KUKA KRL program: EPS_2_251806_MH45A_A_20260213065140.src

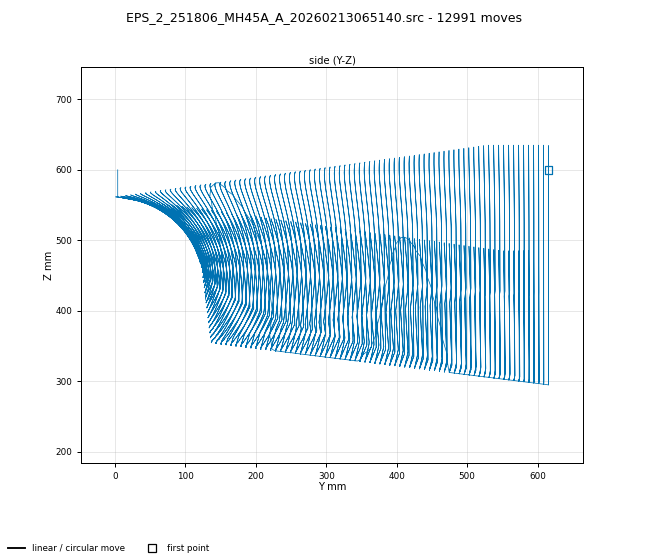
[picture p0: tool path of EPS_2_251806_MH45A_A_20260213065140.src, 12991 of 12993 moves have a stored position in this frame; points joined in program order, loops and branches not executed]
&ACCESS RVP
&REL 4
&COMMENT QRS 19112012
&PARAM EDITMASK = *
DEF PART()
EXT BAS (BAS_COMMAND :IN,REAL :IN )
INT I
BAS (#INITMOV,0 )

;KUKA QRS Post kuka4.cps  Date:22-06-2017 !

File_ID=3032

QRS_PRE_INIT()

;Init var - Until changes are made in qrs_pre_init
Outlet_Square_prg=0
Inlet_1_Square_prg=0
Inlet_2_Square_prg=0
Inlet_3_Square_prg=0
Inlet_4_Square_prg=0
Inlet_5_Square_prg=0

Outlet_1={X 0.000, Y 530.070, Z 534.500, B 0.000, E1 0.000 }
Inlet_1={X 0.000, Y 547.890, Z 284.500, B 0.000, E1 180.000 }
Outlet_1_type=201
Inlet_1_type=201
;QRS#1=Sidecore dimensions
;QRS#2=200-8" PVC SDR 35
;QRS#3=200-8" PVC SDR 35
;QRS#4=
;QRS#5=
;QRS#6=
;QRS#7=
;QRS#8=
;QRS#9=12-08 PSX
;QRS#10=12-08 PSX
;QRS#11=
;QRS#12=
;QRS#13=
;QRS#14=
;QRS#15=
;QRS#16=1220x127x914 3'
;QRS#17=EPS Height
;QRS#18=635
;QRS#19=*
;QRS#20= UPDATED VERSION 22-06-2017
;QRS#21=*
Outlet_Square=0100
Inlet_1_Square=0100
Inlet_2_Square=0
Inlet_3_Square=0
Inlet_4_Square=0
Inlet_5_Square=0
Mill_Square=1
Outlet_Square_Prg=204
Inlet_1_Square_prg=204

QRS_INIT()

$ADVANCE=5

; T1
PTP {E1 173.65,E2 173.65}
PTP {X 0,Y 615.429,A -85,B 0,C 180,E1 173.65,E2 173.65,E3 0,E4 0,E5 0,E6 0}
QRS_SPEED_INIT()
LIN {X 0,Y 615.429,Z 600,A -85,B 0,C 180,E1 173.65,E2 173.65,E3 0,E4 0,E5 0,E6 0} C_VEL
LIN {X 0,Y 615.429,Z 304.876,A -85,B 0,C 180,E1 173.65,E2 173.65} C_VEL
LIN {X 0,Y 615.429,Z 296.697,A -85,B 0,C 180,E1 173.65,E2 173.65} C_VEL
LIN {X 0,Y 615.425,Z 294.697,A -85,B 0,C 180,E1 173.464,E2 173.464} C_VEL
LIN {X 0,Y 615.464,Z 294.694,A -85,B 0,C 180,E1 170.801,E2 170.801} C_VEL
LIN {X 0,Y 615.465,Z 294.699,A -85,B 0,C 180,E1 168.139,E2 168.139} C_VEL
LIN {X 0,Y 615.424,Z 294.696,A -85,B 0,C 180,E1 165.449,E2 165.449} C_VEL
LIN {X 0,Y 615.48,Z 294.694,A -85,B 0,C 180,E1 162.729,E2 162.729} C_VEL
LIN {X 0,Y 615.442,Z 294.698,A -85,B 0,C 180,E1 159.966,E2 159.966} C_VEL
LIN {X 0,Y 615.425,Z 294.697,A -85,B 0,C 180,E1 157.666,E2 157.666} C_VEL
LIN {X 0,Y 615.425,Z 294.698,A -85,B 0,C 180,E1 155.725,E2 155.725} C_VEL
LIN {X 0,Y 615.424,Z 294.697,A -85,B 0,C 180,E1 153.553,E2 153.553} C_VEL
LIN {X 0,Y 615.493,Z 294.698,A -85,B 0,C 180,E1 150.594,E2 150.594} C_VEL
LIN {X 0,Y 615.472,Z 294.699,A -85,B 0,C 180,E1 148.314,E2 148.314} C_VEL
LIN {X 0,Y 615.436,Z 294.698,A -85,B 0,C 180,E1 145.975,E2 145.975} C_VEL
LIN {X 0,Y 615.423,Z 294.697,A -85,B 0,C 180,E1 143.571,E2 143.571} C_VEL
LIN {X 0,Y 615.464,Z 294.695,A -85,B 0,C 180,E1 140.939,E2 140.939} C_VEL
LIN {X 0,Y 615.495,Z 294.7,A -85,B 0,C 180,E1 138.527,E2 138.527} C_VEL
LIN {X 0,Y 615.426,Z 294.697,A -85,B 0,C 180,E1 135.845,E2 135.845} C_VEL
LIN {X 0,Y 615.459,Z 294.695,A -85,B 0,C 180,E1 133.044,E2 133.044} C_VEL
LIN {X 0,Y 615.437,Z 294.698,A -85,B 0,C 180,E1 130.083,E2 130.083} C_VEL
LIN {X 0,Y 615.429,Z 294.698,A -85,B 0,C 180,E1 128.005,E2 128.005} C_VEL
LIN {X 0,Y 615.42,Z 294.697,A -85,B 0,C 180,E1 125.62,E2 125.62} C_VEL
LIN {X 0,Y 615.445,Z 294.695,A -85,B 0,C 180,E1 123.238,E2 123.238} C_VEL
LIN {X 0,Y 615.486,Z 294.694,A -85,B 0,C 180,E1 120.919,E2 120.919} C_VEL
LIN {X 0,Y 615.465,Z 294.699,A -85,B 0,C 180,E1 118.446,E2 118.446} C_VEL
LIN {X 0,Y 615.463,Z 294.699,A -85,B 0,C 180,E1 116.445,E2 116.445} C_VEL
LIN {X 0,Y 615.424,Z 294.698,A -85,B 0,C 180,E1 113.994,E2 113.994} C_VEL
LIN {X 0,Y 615.433,Z 294.698,A -85,B 0,C 180,E1 112.138,E2 112.138} C_VEL
LIN {X 0,Y 615.425,Z 294.698,A -85,B 0,C 180,E1 110.034,E2 110.034} C_VEL
LIN {X 0,Y 615.423,Z 294.698,A -85,B 0,C 180,E1 107.959,E2 107.959} C_VEL
LIN {X 0,Y 615.422,Z 294.697,A -85,B 0,C 180,E1 105.907,E2 105.907} C_VEL
LIN {X 0,Y 615.458,Z 294.696,A -85,B 0,C 180,E1 103.202,E2 103.202} C_VEL
LIN {X 0,Y 615.498,Z 294.906,A -85,B 0,C 180,E1 102.676,E2 102.676} C_VEL
LIN {X 0,Y 615.497,Z 295.813,A -85,B 0,C 180,E1 102.572,E2 102.572} C_VEL
LIN {X 0,Y 615.497,Z 381.802,A -85,B 0,C 180,E1 101.526,E2 101.526} C_VEL
LIN {X 0,Y 615.498,Z 394.745,A -85,B 0,C 180,E1 101.234,E2 101.234} C_VEL
LIN {X 0,Y 615.498,Z 407.738,A -85,B 0,C 180,E1 100.8,E2 100.8} C_VEL
LIN {X 0,Y 615.496,Z 419.198,A -85,B 0,C 180,E1 100.277,E2 100.277} C_VEL
LIN {X 0,Y 615.492,Z 430.579,A -85,B 0,C 180,E1 99.613,E2 99.613} C_VEL
LIN {X 0,Y 615.498,Z 440.825,A -85,B 0,C 180,E1 98.867,E2 98.867} C_VEL
LIN {X 0,Y 615.499,Z 450.035,A -85,B 0,C 180,E1 98.04,E2 98.04} C_VEL
LIN {X 0,Y 615.499,Z 458.893,A -85,B 0,C 180,E1 97.057,E2 97.057} C_VEL
LIN {X 0,Y 615.497,Z 466.124,A -85,B 0,C 180,E1 96.063,E2 96.063} C_VEL
LIN {X 0,Y 615.497,Z 470.958,A -85,B 0,C 180,E1 95.241,E2 95.241} C_VEL
LIN {X 0,Y 615.494,Z 475.658,A -85,B 0,C 180,E1 94.256,E2 94.256} C_VEL
LIN {X 0,Y 615.494,Z 479.255,A -85,B 0,C 180,E1 93.273,E2 93.273} C_VEL
LIN {X 0,Y 615.496,Z 481.115,A -85,B 0,C 180,E1 92.618,E2 92.618} C_VEL
LIN {X 0,Y 615.499,Z 482.533,A -85,B 0,C 180,E1 91.963,E2 91.963} C_VEL
LIN {X 0,Y 615.496,Z 484.142,A -85,B 0,C 180,E1 90.654,E2 90.654} C_VEL
LIN {X 0,Y 615.495,Z 484.384,A -85,B 0,C 180,E1 90,E2 90} C_VEL
LIN {X 0,Y 615.495,Z 484.206,A -85,B 0,C 180,E1 89.346,E2 89.346} C_VEL
LIN {X 0,Y 615.499,Z 482.682,A -85,B 0,C 180,E1 88.037,E2 88.037} C_VEL
LIN {X 0,Y 615.498,Z 481.341,A -85,B 0,C 180,E1 87.382,E2 87.382} C_VEL
LIN {X 0,Y 615.496,Z 478.494,A -85,B 0,C 180,E1 86.399,E2 86.399} C_VEL
LIN {X 0,Y 615.498,Z 474.634,A -85,B 0,C 180,E1 85.416,E2 85.416} C_VEL
LIN {X 0,Y 615.498,Z 469.652,A -85,B 0,C 180,E1 84.43,E2 84.43} C_VEL
LIN {X 0,Y 615.496,Z 463.208,A -85,B 0,C 180,E1 83.418,E2 83.418} C_VEL
LIN {X 0,Y 615.497,Z 455.538,A -85,B 0,C 180,E1 82.455,E2 82.455} C_VEL
LIN {X 0,Y 615.498,Z 445.76,A -85,B 0,C 180,E1 81.464,E2 81.464} C_VEL
LIN {X 0,Y 615.498,Z 435.495,A -85,B 0,C 180,E1 80.636,E2 80.636} C_VEL
LIN {X 0,Y 615.495,Z 423.932,A -85,B 0,C 180,E1 79.889,E2 79.889} C_VEL
LIN {X 0,Y 615.499,Z 412.024,A -85,B 0,C 180,E1 79.291,E2 79.291} C_VEL
LIN {X 0,Y 615.498,Z 399.164,A -85,B 0,C 180,E1 78.807,E2 78.807} C_VEL
LIN {X 0,Y 615.497,Z 386.566,A -85,B 0,C 180,E1 78.474,E2 78.474} C_VEL
LIN {X 0,Y 615.498,Z 373.45,A -85,B 0,C 180,E1 78.265,E2 78.265} C_VEL
LIN {X 0,Y 615.498,Z 295.937,A -85,B 0,C 180,E1 77.345,E2 77.345} C_VEL
LIN {X 0,Y 615.498,Z 294.856,A -85,B 0,C 180,E1 77.219,E2 77.219} C_VEL
LIN {X 0,Y 615.454,Z 294.698,A -85,B 0,C 180,E1 74.773,E2 74.773} C_VEL
LIN {X 0,Y 615.447,Z 294.698,A -85,B 0,C 180,E1 72.729,E2 72.729} C_VEL
LIN {X 0,Y 615.436,Z 294.699,A -85,B 0,C 180,E1 70.661,E2 70.661} C_VEL
LIN {X 0,Y 615.43,Z 294.698,A -85,B 0,C 180,E1 68.566,E2 68.566} C_VEL
LIN {X 0,Y 615.422,Z 294.698,A -85,B 0,C 180,E1 66.441,E2 66.441} C_VEL
LIN {X 0,Y 615.414,Z 294.699,A -85,B 0,C 180,E1 64.281,E2 64.281} C_VEL
LIN {X 0,Y 615.415,Z 294.699,A -85,B 0,C 180,E1 62.082,E2 62.082} C_VEL
LIN {X 0,Y 615.428,Z 294.699,A -85,B 0,C 180,E1 59.837,E2 59.837} C_VEL
LIN {X 0,Y 615.459,Z 294.7,A -85,B 0,C 180,E1 57.541,E2 57.541} C_VEL
LIN {X 0,Y 615.498,Z 294.697,A -85,B 0,C 180,E1 55.186,E2 55.186} C_VEL
LIN {X 0,Y 615.44,Z 294.697,A -85,B 0,C 180,E1 52.755,E2 52.755} C_VEL
LIN {X 0,Y 615.416,Z 294.698,A -85,B 0,C 180,E1 50.245,E2 50.245} C_VEL
LIN {X 0,Y 615.454,Z 294.699,A -85,B 0,C 180,E1 47.645,E2 47.645} C_VEL
LIN {X 0,Y 615.454,Z 294.697,A -85,B 0,C 180,E1 44.929,E2 44.929} C_VEL
LIN {X 0,Y 615.467,Z 294.697,A -85,B 0,C 180,E1 43.046,E2 43.046} C_VEL
LIN {X 0,Y 615.425,Z 294.697,A -85,B 0,C 180,E1 40.612,E2 40.612} C_VEL
LIN {X 0,Y 615.428,Z 294.699,A -85,B 0,C 180,E1 38.006,E2 38.006} C_VEL
LIN {X 0,Y 615.468,Z 294.7,A -85,B 0,C 180,E1 35.617,E2 35.617} C_VEL
LIN {X 0,Y 615.483,Z 294.697,A -85,B 0,C 180,E1 33.237,E2 33.237} C_VEL
LIN {X 0,Y 615.445,Z 294.697,A -85,B 0,C 180,E1 30.922,E2 30.922} C_VEL
LIN {X 0,Y 615.419,Z 294.698,A -85,B 0,C 180,E1 28.44,E2 28.44} C_VEL
LIN {X 0,Y 615.419,Z 294.698,A -85,B 0,C 180,E1 26.447,E2 26.447} C_VEL
LIN {X 0,Y 615.435,Z 294.699,A -85,B 0,C 180,E1 24,E2 24} C_VEL
LIN {X 0,Y 615.498,Z 294.698,A -85,B 0,C 180,E1 21.432,E2 21.432} C_VEL
LIN {X 0,Y 615.421,Z 294.697,A -85,B 0,C 180,E1 18.589,E2 18.589} C_VEL
LIN {X 0,Y 615.42,Z 294.698,A -85,B 0,C 180,E1 16.413,E2 16.413} C_VEL
LIN {X 0,Y 615.451,Z 294.7,A -85,B 0,C 180,E1 13.875,E2 13.875} C_VEL
LIN {X 0,Y 615.464,Z 294.695,A -85,B 0,C 180,E1 11.194,E2 11.194} C_VEL
LIN {X 0,Y 615.421,Z 294.697,A -85,B 0,C 180,E1 8.538,E2 8.538} C_VEL
LIN {X 0,Y 615.454,Z 294.7,A -85,B 0,C 180,E1 5.899,E2 5.899} C_VEL
LIN {X 0,Y 615.469,Z 294.695,A -85,B 0,C 180,E1 3.273,E2 3.273} C_VEL
LIN {X 0,Y 615.422,Z 294.697,A -85,B 0,C 180,E1 0.654,E2 0.654} C_VEL
LIN {X 0,Y 615.45,Z 294.699,A -85,B 0,C 180,E1 -1.963,E2 -1.963} C_VEL
LIN {X 0,Y 615.483,Z 294.694,A -85,B 0,C 180,E1 -4.585,E2 -4.585} C_VEL
LIN {X 0,Y 615.423,Z 294.697,A -85,B 0,C 180,E1 -7.216,E2 -7.216} C_VEL
LIN {X 0,Y 615.425,Z 294.696,A -85,B 0,C 180,E1 -9.2,E2 -9.2} C_VEL
LIN {X 0,Y 615.424,Z 294.697,A -85,B 0,C 180,E1 -11.194,E2 -11.194} C_VEL
LIN {X 0,Y 615.424,Z 294.696,A -85,B 0,C 180,E1 -13.203,E2 -13.203} C_VEL
LIN {X 0,Y 615.422,Z 294.697,A -85,B 0,C 180,E1 -15.228,E2 -15.228} C_VEL
LIN {X 0,Y 615.422,Z 294.697,A -85,B 0,C 180,E1 -17.272,E2 -17.272} C_VEL
LIN {X 0,Y 615.423,Z 294.697,A -85,B 0,C 180,E1 -19.34,E2 -19.34} C_VEL
LIN {X 0,Y 615.425,Z 294.697,A -85,B 0,C 180,E1 -21.434,E2 -21.434} C_VEL
LIN {X 0,Y 615.473,Z 294.699,A -85,B 0,C 180,E1 -24.008,E2 -24.008} C_VEL
LIN {X 0,Y 615.486,Z 294.694,A -85,B 0,C 180,E1 -26.444,E2 -26.444} C_VEL
LIN {X 0,Y 615.456,Z 294.694,A -85,B 0,C 180,E1 -28.66,E2 -28.66} C_VEL
LIN {X 0,Y 615.427,Z 294.696,A -85,B 0,C 180,E1 -31.078,E2 -31.078} C_VEL
LIN {X 0,Y 615.425,Z 294.697,A -85,B 0,C 180,E1 -33.24,E2 -33.24} C_VEL
LIN {X 0,Y 615.458,Z 294.7,A -85,B 0,C 180,E1 -35.831,E2 -35.831} C_VEL
LIN {X 0,Y 615.487,Z 294.702,A -85,B 0,C 180,E1 -38.069,E2 -38.069} C_VEL
LIN {X 0,Y 615.455,Z 294.694,A -85,B 0,C 180,E1 -40.609,E2 -40.609} C_VEL
LIN {X 0,Y 615.427,Z 294.696,A -85,B 0,C 180,E1 -43.042,E2 -43.042} C_VEL
LIN {X 0,Y 615.426,Z 294.696,A -85,B 0,C 180,E1 -45.074,E2 -45.074} C_VEL
LIN {X 0,Y 615.45,Z 294.698,A -85,B 0,C 180,E1 -47.645,E2 -47.645} C_VEL
LIN {X 0,Y 615.491,Z 294.693,A -85,B 0,C 180,E1 -50.251,E2 -50.251} C_VEL
LIN {X 0,Y 615.437,Z 294.695,A -85,B 0,C 180,E1 -52.755,E2 -52.755} C_VEL
LIN {X 0,Y 615.427,Z 294.697,A -85,B 0,C 180,E1 -55.182,E2 -55.182} C_VEL
LIN {X 0,Y 615.46,Z 294.699,A -85,B 0,C 180,E1 -57.674,E2 -57.674} C_VEL
LIN {X 0,Y 615.447,Z 294.694,A -85,B 0,C 180,E1 -60.592,E2 -60.592} C_VEL
LIN {X 0,Y 615.426,Z 294.696,A -85,B 0,C 180,E1 -62.967,E2 -62.967} C_VEL
LIN {X 0,Y 615.497,Z 294.938,A -85,B 0,C 180,E1 -64.058,E2 -64.058} C_VEL
LIN {X 0,Y 615.487,Z 314.816,A -85,B 0,C 180,E1 -66.218,E2 -66.218} C_VEL
LIN {X 0,Y 615.493,Z 342.158,A -85,B 0,C 180,E1 -69.095,E2 -69.095} C_VEL
LIN {X 0,Y 615.484,Z 369.157,A -85,B 0,C 180,E1 -71.882,E2 -71.882} C_VEL
LIN {X 0,Y 615.477,Z 395.91,A -85,B 0,C 180,E1 -74.604,E2 -74.604} C_VEL
LIN {X 0,Y 615.498,Z 420.869,A -85,B 0,C 180,E1 -77.093,E2 -77.093} C_VEL
LIN {X 0,Y 615.486,Z 530.842,A -85,B 0,C 180,E1 -78.411,E2 -78.411} C_VEL
LIN {X 0,Y 615.499,Z 543.349,A -85,B 0,C 180,E1 -78.682,E2 -78.682} C_VEL
LIN {X 0,Y 615.496,Z 556.5,A -85,B 0,C 180,E1 -79.109,E2 -79.109} C_VEL
LIN {X 0,Y 615.482,Z 568.481,A -85,B 0,C 180,E1 -79.639,E2 -79.639} C_VEL
LIN {X 0,Y 615.487,Z 579.998,A -85,B 0,C 180,E1 -80.304,E2 -80.304} C_VEL
LIN {X 0,Y 615.499,Z 590.343,A -85,B 0,C 180,E1 -81.05,E2 -81.05} C_VEL
LIN {X 0,Y 615.497,Z 598.813,A -85,B 0,C 180,E1 -81.794,E2 -81.794} C_VEL
LIN {X 0,Y 615.498,Z 606.607,A -85,B 0,C 180,E1 -82.62,E2 -82.62} C_VEL
LIN {X 0,Y 615.496,Z 614.204,A -85,B 0,C 180,E1 -83.608,E2 -83.608} C_VEL
LIN {X 0,Y 615.498,Z 621.205,A -85,B 0,C 180,E1 -84.759,E2 -84.759} C_VEL
LIN {X 0,Y 615.493,Z 625.852,A -85,B 0,C 180,E1 -85.744,E2 -85.744} C_VEL
LIN {X 0,Y 615.495,Z 629.399,A -85,B 0,C 180,E1 -86.727,E2 -86.727} C_VEL
LIN {X 0,Y 615.497,Z 631.233,A -85,B 0,C 180,E1 -87.382,E2 -87.382} C_VEL
LIN {X 0,Y 615.497,Z 632.608,A -85,B 0,C 180,E1 -88.037,E2 -88.037} C_VEL
LIN {X 0,Y 615.496,Z 634.174,A -85,B 0,C 180,E1 -89.346,E2 -89.346} C_VEL
LIN {X 0,Y 615.494,Z 634.389,A -85,B 0,C 180,E1 -90,E2 -90} C_VEL
LIN {X 0,Y 615.496,Z 633.58,A -85,B 0,C 180,E1 -91.309,E2 -91.309} C_VEL
LIN {X 0,Y 615.497,Z 632.608,A -85,B 0,C 180,E1 -91.963,E2 -91.963} C_VEL
LIN {X 0,Y 615.497,Z 631.233,A -85,B 0,C 180,E1 -92.618,E2 -92.618} C_VEL
LIN {X 0,Y 615.496,Z 628.35,A -85,B 0,C 180,E1 -93.601,E2 -93.601} C_VEL
LIN {X 0,Y 615.498,Z 624.442,A -85,B 0,C 180,E1 -94.584,E2 -94.584} C_VEL
LIN {X 0,Y 615.499,Z 619.405,A -85,B 0,C 180,E1 -95.57,E2 -95.57} C_VEL
LIN {X 0,Y 615.497,Z 612.869,A -85,B 0,C 180,E1 -96.583,E2 -96.583} C_VEL
LIN {X 0,Y 615.497,Z 605.134,A -85,B 0,C 180,E1 -97.545,E2 -97.545} C_VEL
LIN {X 0,Y 615.498,Z 597.047,A -85,B 0,C 180,E1 -98.371,E2 -98.371} C_VEL
LIN {X 0,Y 615.499,Z 587.17,A -85,B 0,C 180,E1 -99.198,E2 -99.198} C_VEL
LIN {X 0,Y 615.488,Z 575.985,A -85,B 0,C 180,E1 -99.945,E2 -99.945} C_VEL
LIN {X 0,Y 615.486,Z 565.027,A -85,B 0,C 180,E1 -100.527,E2 -100.527} C_VEL
LIN {X 0,Y 615.499,Z 552.418,A -85,B 0,C 180,E1 -101.042,E2 -101.042} C_VEL
LIN {X 0,Y 615.498,Z 540.072,A -85,B 0,C 180,E1 -101.401,E2 -101.401} C_VEL
LIN {X 0,Y 615.484,Z 526.483,A -85,B 0,C 180,E1 -101.652,E2 -101.652} C_VEL
LIN {X 0,Y 615.498,Z 420.869,A -85,B 0,C 180,E1 -102.907,E2 -102.907} C_VEL
LIN {X 0,Y 615.477,Z 395.91,A -85,B 0,C 180,E1 -105.396,E2 -105.396} C_VEL
LIN {X 0,Y 615.484,Z 369.157,A -85,B 0,C 180,E1 -108.118,E2 -108.118} C_VEL
LIN {X 0,Y 615.493,Z 342.159,A -85,B 0,C 180,E1 -110.905,E2 -110.905} C_VEL
LIN {X 0,Y 615.487,Z 314.813,A -85,B 0,C 180,E1 -113.782,E2 -113.782} C_VEL
LIN {X 0,Y 615.495,Z 294.938,A -85,B 0,C 180,E1 -115.942,E2 -115.942} C_VEL
LIN {X 0,Y 615.43,Z 294.695,A -85,B 0,C 180,E1 -117.179,E2 -117.179} C_VEL
LIN {X 0,Y 615.494,Z 294.692,A -85,B 0,C 180,E1 -119.795,E2 -119.795} C_VEL
LIN {X 0,Y 615.448,Z 294.698,A -85,B 0,C 180,E1 -122.459,E2 -122.459} C_VEL
LIN {X 0,Y 615.428,Z 294.696,A -85,B 0,C 180,E1 -124.818,E2 -124.818} C_VEL
LIN {X 0,Y 615.437,Z 294.695,A -85,B 0,C 180,E1 -127.245,E2 -127.245} C_VEL
LIN {X 0,Y 615.485,Z 294.7,A -85,B 0,C 180,E1 -130.089,E2 -130.089} C_VEL
LIN {X 0,Y 615.451,Z 294.698,A -85,B 0,C 180,E1 -132.355,E2 -132.355} C_VEL
LIN {X 0,Y 615.427,Z 294.696,A -85,B 0,C 180,E1 -134.926,E2 -134.926} C_VEL
LIN {X 0,Y 615.428,Z 294.696,A -85,B 0,C 180,E1 -136.957,E2 -136.957} C_VEL
LIN {X 0,Y 615.456,Z 294.694,A -85,B 0,C 180,E1 -139.391,E2 -139.391} C_VEL
LIN {X 0,Y 615.479,Z 294.702,A -85,B 0,C 180,E1 -141.988,E2 -141.988} C_VEL
LIN {X 0,Y 615.443,Z 294.698,A -85,B 0,C 180,E1 -144.381,E2 -144.381} C_VEL
LIN {X 0,Y 615.426,Z 294.696,A -85,B 0,C 180,E1 -146.76,E2 -146.76} C_VEL
LIN {X 0,Y 615.435,Z 294.695,A -85,B 0,C 180,E1 -149.077,E2 -149.077} C_VEL
LIN {X 0,Y 615.484,Z 294.693,A -85,B 0,C 180,E1 -151.548,E2 -151.548} C_VEL
LIN {X 0,Y 615.446,Z 294.698,A -85,B 0,C 180,E1 -154.282,E2 -154.282} C_VEL
LIN {X 0,Y 615.434,Z 294.697,A -85,B 0,C 180,E1 -156.441,E2 -156.441} C_VEL
LIN {X 0,Y 615.428,Z 294.697,A -85,B 0,C 180,E1 -158.566,E2 -158.566} C_VEL
LIN {X 0,Y 615.426,Z 294.696,A -85,B 0,C 180,E1 -160.66,E2 -160.66} C_VEL
LIN {X 0,Y 615.471,Z 294.694,A -85,B 0,C 180,E1 -163.413,E2 -163.413} C_VEL
LIN {X 0,Y 615.453,Z 294.699,A -85,B 0,C 180,E1 -166.125,E2 -166.125} C_VEL
LIN {X 0,Y 615.451,Z 294.698,A -85,B 0,C 180,E1 -168.138,E2 -168.138} C_VEL
LIN {X 0,Y 615.45,Z 294.698,A -85,B 0,C 180,E1 -170.137,E2 -170.137} C_VEL
LIN {X 0,Y 615.45,Z 294.698,A -85,B 0,C 180,E1 -172.124,E2 -172.124} C_VEL
LIN {X 0,Y 615.451,Z 294.699,A -85,B 0,C 180,E1 -174.101,E2 -174.101} C_VEL
LIN {X 0,Y 615.453,Z 294.699,A -85,B 0,C 180,E1 -176.071,E2 -176.071} C_VEL
LIN {X 0,Y 615.455,Z 294.699,A -85,B 0,C 180,E1 -178.037,E2 -178.037} C_VEL
LIN {X 0,Y 615.425,Z 294.696,A -85,B 0,C 180,E1 -180.654,E2 -180.654} C_VEL
LIN {X 0,Y 615.469,Z 294.694,A -85,B 0,C 180,E1 -183.273,E2 -183.273} C_VEL
LIN {X 0,Y 615.465,Z 294.699,A -85,B 0,C 180,E1 -185.899,E2 -185.899} C_VEL
LIN {X 0,Y 615.425,Z 294.697,A -85,B 0,C 180,E1 -186.536,E2 -186.536} C_VEL
LIN {X 0,Y 614.774,Z 294.843,A -85,B 0,C 180,E1 -187.082,E2 -187.082} C_VEL
LIN {X 0,Y 611.963,Z 295.255,A -85,B 0,C 180,E1 -187.968,E2 -187.968} C_VEL
LIN {X 0,Y 609.573,Z 295.565,A -85,B 0,C 180,E1 -188.681,E2 -188.681} C_VEL
LIN {X 0,Y 608.533,Z 295.683,A -85,B 0,C 180,E1 -189.231,E2 -189.231} C_VEL
LIN {X 0,Y 608.441,Z 295.693,A -85,B 0,C 180,E1 -189.417,E2 -189.417} C_VEL
LIN {X 0,Y 608.434,Z 295.694,A -85,B 0,C 180,E1 -192,E2 -192} C_VEL
LIN {X 0,Y 608.4,Z 295.694,A -85,B 0,C 180,E1 -194.722,E2 -194.722} C_VEL
LIN {X 0,Y 608.438,Z 295.698,A -85,B 0,C 180,E1 -197.477,E2 -197.477} C_VEL
LIN {X 0,Y 608.413,Z 295.693,A -85,B 0,C 180,E1 -200.276,E2 -200.276} C_VEL
LIN {X 0,Y 608.42,Z 295.691,A -85,B 0,C 180,E1 -202.47,E2 -202.47} C_VEL
LIN {X 0,Y 608.436,Z 295.696,A -85,B 0,C 180,E1 -205.302,E2 -205.302} C_VEL
LIN {X 0,Y 608.426,Z 295.701,A -85,B 0,C 180,E1 -207.519,E2 -207.519} C_VEL
LIN {X 0,Y 608.417,Z 295.694,A -85,B 0,C 180,E1 -209.965,E2 -209.965} C_VEL
LIN {X 0,Y 608.407,Z 295.693,A -85,B 0,C 180,E1 -212.516,E2 -212.516} C_VEL
LIN {X 0,Y 608.41,Z 295.694,A -85,B 0,C 180,E1 -214.902,E2 -214.902} C_VEL
LIN {X 0,Y 608.438,Z 295.694,A -85,B 0,C 180,E1 -217.749,E2 -217.749} C_VEL
LIN {X 0,Y 608.396,Z 295.694,A -85,B 0,C 180,E1 -220.324,E2 -220.324} C_VEL
LIN {X 0,Y 608.394,Z 295.694,A -85,B 0,C 180,E1 -222.329,E2 -222.329} C_VEL
LIN {X 0,Y 608.404,Z 295.693,A -85,B 0,C 180,E1 -224.26,E2 -224.26} C_VEL
LIN {X 0,Y 608.427,Z 295.695,A -85,B 0,C 180,E1 -227.039,E2 -227.039} C_VEL
LIN {X 0,Y 608.435,Z 295.695,A -85,B 0,C 180,E1 -229.696,E2 -229.696} C_VEL
LIN {X 0,Y 608.401,Z 295.693,A -85,B 0,C 180,E1 -232.25,E2 -232.25} C_VEL
LIN {X 0,Y 608.454,Z 295.693,A -85,B 0,C 180,E1 -235.094,E2 -235.094} C_VEL
LIN {X 0,Y 608.428,Z 295.692,A -85,B 0,C 180,E1 -237.904,E2 -237.904} C_VEL
LIN {X 0,Y 608.41,Z 295.693,A -85,B 0,C 180,E1 -240.218,E2 -240.218} C_VEL
LIN {X 0,Y 608.436,Z 295.691,A -85,B 0,C 180,E1 -242.801,E2 -242.801} C_VEL
LIN {X 0,Y 608.429,Z 295.699,A -85,B 0,C 180,E1 -245.428,E2 -245.428} C_VEL
LIN {X 0,Y 608.421,Z 295.691,A -85,B 0,C 180,E1 -248.307,E2 -248.307} C_VEL
LIN {X 0,Y 608.406,Z 295.693,A -85,B 0,C 180,E1 -250.428,E2 -250.428} C_VEL
LIN {X 0,Y 608.413,Z 295.692,A -85,B 0,C 180,E1 -252.523,E2 -252.523} C_VEL
LIN {X 0,Y 608.426,Z 295.701,A -85,B 0,C 180,E1 -255.279,E2 -255.279} C_VEL
LIN {X 0,Y 608.496,Z 295.84,A -85,B 0,C 180,E1 -257.197,E2 -257.197} C_VEL
LIN {X 0,Y 608.589,Z 296.919,A -85,B 0,C 180,E1 -257.305,E2 -257.305} C_VEL
LIN {X 0,Y 608.558,Z 380.807,A -85,B 0,C 180,E1 -258.319,E2 -258.319} C_VEL
LIN {X 0,Y 608.538,Z 394.124,A -85,B 0,C 180,E1 -258.614,E2 -258.614} C_VEL
LIN {X 0,Y 608.529,Z 407.354,A -85,B 0,C 180,E1 -259.055,E2 -259.055} C_VEL
LIN {X 0,Y 608.508,Z 419.373,A -85,B 0,C 180,E1 -259.604,E2 -259.604} C_VEL
LIN {X 0,Y 608.506,Z 430.793,A -85,B 0,C 180,E1 -260.276,E2 -260.276} C_VEL
LIN {X 0,Y 608.474,Z 441.086,A -85,B 0,C 180,E1 -261.03,E2 -261.03} C_VEL
LIN {X 0,Y 608.464,Z 450.351,A -85,B 0,C 180,E1 -261.866,E2 -261.866} C_VEL
LIN {X 0,Y 608.466,Z 459.324,A -85,B 0,C 180,E1 -262.868,E2 -262.868} C_VEL
LIN {X 0,Y 608.444,Z 466.556,A -85,B 0,C 180,E1 -263.867,E2 -263.867} C_VEL
LIN {X 0,Y 608.462,Z 471.435,A -85,B 0,C 180,E1 -264.698,E2 -264.698} C_VEL
LIN {X 0,Y 608.439,Z 476.179,A -85,B 0,C 180,E1 -265.694,E2 -265.694} C_VEL
LIN {X 0,Y 608.425,Z 479.812,A -85,B 0,C 180,E1 -266.689,E2 -266.689} C_VEL
LIN {X 0,Y 608.425,Z 481.691,A -85,B 0,C 180,E1 -267.352,E2 -267.352} C_VEL
LIN {X 0,Y 608.444,Z 483.127,A -85,B 0,C 180,E1 -268.014,E2 -268.014} C_VEL
LIN {X 0,Y 608.439,Z 484.752,A -85,B 0,C 180,E1 -269.338,E2 -269.338} C_VEL
LIN {X 0,Y 608.435,Z 484.995,A -85,B 0,C 180,E1 -270,E2 -270} C_VEL
LIN {X 0,Y 608.438,Z 484.815,A -85,B 0,C 180,E1 -270.662,E2 -270.662} C_VEL
LIN {X 0,Y 608.444,Z 483.276,A -85,B 0,C 180,E1 -271.986,E2 -271.986} C_VEL
LIN {X 0,Y 608.426,Z 481.919,A -85,B 0,C 180,E1 -272.648,E2 -272.648} C_VEL
LIN {X 0,Y 608.449,Z 479.042,A -85,B 0,C 180,E1 -273.642,E2 -273.642} C_VEL
LIN {X 0,Y 608.433,Z 475.143,A -85,B 0,C 180,E1 -274.638,E2 -274.638} C_VEL
LIN {X 0,Y 608.45,Z 470.113,A -85,B 0,C 180,E1 -275.634,E2 -275.634} C_VEL
LIN {X 0,Y 608.441,Z 463.796,A -85,B 0,C 180,E1 -276.633,E2 -276.633} C_VEL
LIN {X 0,Y 608.475,Z 455.879,A -85,B 0,C 180,E1 -277.633,E2 -277.633} C_VEL
LIN {X 0,Y 608.472,Z 446.037,A -85,B 0,C 180,E1 -278.636,E2 -278.636} C_VEL
LIN {X 0,Y 608.48,Z 435.717,A -85,B 0,C 180,E1 -279.473,E2 -279.473} C_VEL
LIN {X 0,Y 608.492,Z 424.103,A -85,B 0,C 180,E1 -280.229,E2 -280.229} C_VEL
LIN {X 0,Y 608.529,Z 412.86,A -85,B 0,C 180,E1 -280.803,E2 -280.803} C_VEL
LIN {X 0,Y 608.538,Z 401.266,A -85,B 0,C 180,E1 -281.257,E2 -281.257} C_VEL
LIN {X 0,Y 608.539,Z 387.57,A -85,B 0,C 180,E1 -281.639,E2 -281.639} C_VEL
LIN {X 0,Y 608.573,Z 375.305,A -85,B 0,C 180,E1 -281.849,E2 -281.849} C_VEL
LIN {X 0,Y 608.593,Z 297.073,A -85,B 0,C 180,E1 -282.78,E2 -282.78} C_VEL
LIN {X 0,Y 608.507,Z 295.861,A -85,B 0,C 180,E1 -282.888,E2 -282.888} C_VEL
LIN {X 0,Y 608.431,Z 295.692,A -85,B 0,C 180,E1 -285.407,E2 -285.407} C_VEL
LIN {X 0,Y 608.395,Z 295.693,A -85,B 0,C 180,E1 -288.173,E2 -288.173} C_VEL
LIN {X 0,Y 608.44,Z 295.696,A -85,B 0,C 180,E1 -290.982,E2 -290.982} C_VEL
LIN {X 0,Y 608.425,Z 295.696,A -85,B 0,C 180,E1 -293.125,E2 -293.125} C_VEL
LIN {X 0,Y 608.394,Z 295.694,A -85,B 0,C 180,E1 -295.705,E2 -295.705} C_VEL
LIN {X 0,Y 608.404,Z 295.695,A -85,B 0,C 180,E1 -298.269,E2 -298.269} C_VEL
LIN {X 0,Y 608.433,Z 295.692,A -85,B 0,C 180,E1 -301.265,E2 -301.265} C_VEL
LIN {X 0,Y 608.395,Z 295.694,A -85,B 0,C 180,E1 -303.724,E2 -303.724} C_VEL
LIN {X 0,Y 608.424,Z 295.692,A -85,B 0,C 180,E1 -306.093,E2 -306.093} C_VEL
LIN {X 0,Y 608.413,Z 295.701,A -85,B 0,C 180,E1 -308.591,E2 -308.591} C_VEL
LIN {X 0,Y 608.416,Z 295.693,A -85,B 0,C 180,E1 -311.337,E2 -311.337} C_VEL
LIN {X 0,Y 608.417,Z 295.692,A -85,B 0,C 180,E1 -313.873,E2 -313.873} C_VEL
LIN {X 0,Y 608.48,Z 295.694,A -85,B 0,C 180,E1 -316.689,E2 -316.689} C_VEL
LIN {X 0,Y 608.442,Z 295.696,A -85,B 0,C 180,E1 -318.822,E2 -318.822} C_VEL
LIN {X 0,Y 608.396,Z 295.694,A -85,B 0,C 180,E1 -321.406,E2 -321.406} C_VEL
LIN {X 0,Y 608.423,Z 295.692,A -85,B 0,C 180,E1 -323.956,E2 -323.956} C_VEL
LIN {X 0,Y 608.436,Z 295.696,A -85,B 0,C 180,E1 -326.327,E2 -326.327} C_VEL
LIN {X 0,Y 608.435,Z 295.697,A -85,B 0,C 180,E1 -328.733,E2 -328.733} C_VEL
LIN {X 0,Y 608.418,Z 295.691,A -85,B 0,C 180,E1 -331.388,E2 -331.388} C_VEL
LIN {X 0,Y 608.402,Z 295.694,A -85,B 0,C 180,E1 -333.223,E2 -333.223} C_VEL
LIN {X 0,Y 608.405,Z 295.693,A -85,B 0,C 180,E1 -335.427,E2 -335.427} C_VEL
LIN {X 0,Y 608.453,Z 295.694,A -85,B 0,C 180,E1 -338.308,E2 -338.308} C_VEL
LIN {X 0,Y 608.407,Z 295.693,A -85,B 0,C 180,E1 -341.299,E2 -341.299} C_VEL
LIN {X 0,Y 608.415,Z 295.694,A -85,B 0,C 180,E1 -343.905,E2 -343.905} C_VEL
LIN {X 0,Y 608.441,Z 295.696,A -85,B 0,C 180,E1 -346.643,E2 -346.643} C_VEL
LIN {X 0,Y 608.406,Z 295.693,A -85,B 0,C 180,E1 -349.349,E2 -349.349} C_VEL
LIN {X 0,Y 608.402,Z 295.693,A -85,B 0,C 180,E1 -351.363,E2 -351.363} C_VEL
LIN {X 0,Y 608.425,Z 295.695,A -85,B 0,C 180,E1 -354.033,E2 -354.033} C_VEL
LIN {X 0,Y 608.462,Z 295.691,A -85,B 0,C 180,E1 -356.689,E2 -356.689} C_VEL
LIN {X 0,Y 608.401,Z 295.693,A -85,B 0,C 180,E1 -359.338,E2 -359.338} C_VEL
LIN {X 0,Y 608.412,Z 295.692,A -85,B 0,C 180,E1 -361.324,E2 -361.324} C_VEL
LIN {X 0,Y 608.394,Z 295.694,A -85,B 0,C 180,E1 -363.311,E2 -363.311} C_VEL
LIN {X 0,Y 608.425,Z 295.695,A -85,B 0,C 180,E1 -365.967,E2 -365.967} C_VEL
LIN {X 0,Y 608.442,Z 295.693,A -85,B 0,C 180,E1 -368.636,E2 -368.636} C_VEL
LIN {X 0,Y 608.403,Z 295.693,A -85,B 0,C 180,E1 -371.325,E2 -371.325} C_VEL
LIN {X 0,Y 608.443,Z 295.695,A -85,B 0,C 180,E1 -374.011,E2 -374.011} C_VEL
LIN {X 0,Y 608.421,Z 295.693,A -85,B 0,C 180,E1 -376.785,E2 -376.785} C_VEL
LIN {X 0,Y 608.41,Z 295.694,A -85,B 0,C 180,E1 -379.572,E2 -379.572} C_VEL
LIN {X 0,Y 608.469,Z 295.692,A -85,B 0,C 180,E1 -382.406,E2 -382.406} C_VEL
LIN {X 0,Y 608.435,Z 295.694,A -85,B 0,C 180,E1 -384.572,E2 -384.572} C_VEL
LIN {X 0,Y 608.414,Z 295.693,A -85,B 0,C 180,E1 -387.52,E2 -387.52} C_VEL
LIN {X 0,Y 608.47,Z 295.692,A -85,B 0,C 180,E1 -389.974,E2 -389.974} C_VEL
LIN {X 0,Y 608.425,Z 295.691,A -85,B 0,C 180,E1 -392.882,E2 -392.882} C_VEL
LIN {X 0,Y 608.402,Z 295.694,A -85,B 0,C 180,E1 -395.281,E2 -395.281} C_VEL
LIN {X 0,Y 608.46,Z 295.694,A -85,B 0,C 180,E1 -398.241,E2 -398.241} C_VEL
LIN {X 0,Y 608.397,Z 295.694,A -85,B 0,C 180,E1 -401.182,E2 -401.182} C_VEL
LIN {X 0,Y 608.422,Z 295.692,A -85,B 0,C 180,E1 -403.305,E2 -403.305} C_VEL
LIN {X 0,Y 608.462,Z 295.695,A -85,B 0,C 180,E1 -406.131,E2 -406.131} C_VEL
LIN {X 0,Y 608.406,Z 295.693,A -85,B 0,C 180,E1 -408.82,E2 -408.82} C_VEL
LIN {X 0,Y 608.453,Z 295.693,A -85,B 0,C 180,E1 -411.762,E2 -411.762} C_VEL
LIN {X 0,Y 608.416,Z 295.693,A -85,B 0,C 180,E1 -414.721,E2 -414.721} C_VEL
LIN {X 0,Y 608.428,Z 295.693,A -85,B 0,C 180,E1 -417.483,E2 -417.483} C_VEL
LIN {X 0,Y 608.478,Z 295.69,A -85,B 0,C 180,E1 -420.222,E2 -420.222} C_VEL
LIN {X 0,Y 608.399,Z 295.697,A -85,B 0,C 180,E1 -423.224,E2 -423.224} C_VEL
LIN {X 0,Y 608.498,Z 295.939,A -85,B 0,C 180,E1 -423.864,E2 -423.864} C_VEL
LIN {X 0,Y 608.724,Z 300.805,A -85,B 0,C 180,E1 -424.418,E2 -424.418} C_VEL
LIN {X 0,Y 608.656,Z 325.517,A -85,B 0,C 180,E1 -427.082,E2 -427.082} C_VEL
LIN {X 0,Y 608.597,Z 352.244,A -85,B 0,C 180,E1 -429.907,E2 -429.907} C_VEL
LIN {X 0,Y 608.549,Z 379.14,A -85,B 0,C 180,E1 -432.7,E2 -432.7} C_VEL
LIN {X 0,Y 608.515,Z 406.036,A -85,B 0,C 180,E1 -435.452,E2 -435.452} C_VEL
LIN {X 0,Y 608.531,Z 420.908,A -85,B 0,C 180,E1 -436.943,E2 -436.943} C_VEL
LIN {X 0,Y 608.538,Z 530.958,A -85,B 0,C 180,E1 -438.277,E2 -438.277} C_VEL
LIN {X 0,Y 608.545,Z 544.223,A -85,B 0,C 180,E1 -438.572,E2 -438.572} C_VEL
LIN {X 0,Y 608.544,Z 557.333,A -85,B 0,C 180,E1 -439.009,E2 -439.009} C_VEL
LIN {X 0,Y 608.503,Z 568.638,A -85,B 0,C 180,E1 -439.519,E2 -439.519} C_VEL
LIN {X 0,Y 608.48,Z 580.2,A -85,B 0,C 180,E1 -440.191,E2 -440.191} C_VEL
LIN {X 0,Y 608.485,Z 590.596,A -85,B 0,C 180,E1 -440.946,E2 -440.946} C_VEL
LIN {X 0,Y 608.475,Z 599.113,A -85,B 0,C 180,E1 -441.699,E2 -441.699} C_VEL
LIN {X 0,Y 608.471,Z 606.961,A -85,B 0,C 180,E1 -442.534,E2 -442.534} C_VEL
LIN {X 0,Y 608.461,Z 614.287,A -85,B 0,C 180,E1 -443.485,E2 -443.485} C_VEL
LIN {X 0,Y 608.45,Z 619.866,A -85,B 0,C 180,E1 -444.366,E2 -444.366} C_VEL
LIN {X 0,Y 608.432,Z 624.95,A -85,B 0,C 180,E1 -445.362,E2 -445.362} C_VEL
LIN {X 0,Y 608.449,Z 628.896,A -85,B 0,C 180,E1 -446.358,E2 -446.358} C_VEL
LIN {X 0,Y 608.425,Z 631.809,A -85,B 0,C 180,E1 -447.352,E2 -447.352} C_VEL
LIN {X 0,Y 608.442,Z 633.201,A -85,B 0,C 180,E1 -448.014,E2 -448.014} C_VEL
LIN {X 0,Y 608.438,Z 634.783,A -85,B 0,C 180,E1 -449.338,E2 -449.338} C_VEL
LIN {X 0,Y 608.434,Z 635,A -85,B 0,C 180,E1 -450,E2 -450} C_VEL
LIN {X 0,Y 608.448,Z 634.184,A -85,B 0,C 180,E1 -451.324,E2 -451.324} C_VEL
LIN {X 0,Y 608.443,Z 633.201,A -85,B 0,C 180,E1 -451.986,E2 -451.986} C_VEL
LIN {X 0,Y 608.425,Z 631.809,A -85,B 0,C 180,E1 -452.648,E2 -452.648} C_VEL
LIN {X 0,Y 608.449,Z 628.896,A -85,B 0,C 180,E1 -453.642,E2 -453.642} C_VEL
LIN {X 0,Y 608.432,Z 624.95,A -85,B 0,C 180,E1 -454.638,E2 -454.638} C_VEL
LIN {X 0,Y 608.437,Z 618.877,A -85,B 0,C 180,E1 -455.801,E2 -455.801} C_VEL
LIN {X 0,Y 608.462,Z 612.236,A -85,B 0,C 180,E1 -456.799,E2 -456.799} C_VEL
LIN {X 0,Y 608.455,Z 603.99,A -85,B 0,C 180,E1 -457.8,E2 -457.8} C_VEL
LIN {X 0,Y 608.472,Z 595.538,A -85,B 0,C 180,E1 -458.636,E2 -458.636} C_VEL
LIN {X 0,Y 608.471,Z 585.093,A -85,B 0,C 180,E1 -459.473,E2 -459.473} C_VEL
LIN {X 0,Y 608.495,Z 574.759,A -85,B 0,C 180,E1 -460.144,E2 -460.144} C_VEL
LIN {X 0,Y 608.522,Z 563.243,A -85,B 0,C 180,E1 -460.741,E2 -460.741} C_VEL
LIN {X 0,Y 608.533,Z 551.878,A -85,B 0,C 180,E1 -461.192,E2 -461.192} C_VEL
LIN {X 0,Y 608.554,Z 538.362,A -85,B 0,C 180,E1 -461.575,E2 -461.575} C_VEL
LIN {X 0,Y 608.547,Z 525.101,A -85,B 0,C 180,E1 -461.808,E2 -461.808} C_VEL
LIN {X 0,Y 608.531,Z 420.907,A -85,B 0,C 180,E1 -463.057,E2 -463.057} C_VEL
LIN {X 0,Y 608.532,Z 392.588,A -85,B 0,C 180,E1 -465.919,E2 -465.919} C_VEL
LIN {X 0,Y 608.59,Z 364.011,A -85,B 0,C 180,E1 -468.865,E2 -468.865} C_VEL
LIN {X 0,Y 608.624,Z 337.116,A -85,B 0,C 180,E1 -471.685,E2 -471.685} C_VEL
LIN {X 0,Y 608.703,Z 311.369,A -85,B 0,C 180,E1 -474.436,E2 -474.436} C_VEL
LIN {X 0,Y 608.681,Z 296.772,A -85,B 0,C 180,E1 -476.024,E2 -476.024} C_VEL
LIN {X 0,Y 608.47,Z 295.745,A -85,B 0,C 180,E1 -476.195,E2 -476.195} C_VEL
LIN {X 0,Y 608.4,Z 295.694,A -85,B 0,C 180,E1 -479.023,E2 -479.023} C_VEL
LIN {X 0,Y 608.43,Z 295.691,A -85,B 0,C 180,E1 -481.318,E2 -481.318} C_VEL
LIN {X 0,Y 608.444,Z 295.694,A -85,B 0,C 180,E1 -483.731,E2 -483.731} C_VEL
LIN {X 0,Y 608.44,Z 295.699,A -85,B 0,C 180,E1 -486.092,E2 -486.092} C_VEL
LIN {X 0,Y 608.403,Z 295.695,A -85,B 0,C 180,E1 -488.592,E2 -488.592} C_VEL
LIN {X 0,Y 608.426,Z 295.692,A -85,B 0,C 180,E1 -491.338,E2 -491.338} C_VEL
LIN {X 0,Y 608.439,Z 295.694,A -85,B 0,C 180,E1 -494.262,E2 -494.262} C_VEL
LIN {X 0,Y 608.423,Z 295.691,A -85,B 0,C 180,E1 -496.695,E2 -496.695} C_VEL
LIN {X 0,Y 608.398,Z 295.694,A -85,B 0,C 180,E1 -498.819,E2 -498.819} C_VEL
LIN {X 0,Y 608.459,Z 295.694,A -85,B 0,C 180,E1 -501.759,E2 -501.759} C_VEL
LIN {X 0,Y 608.404,Z 295.693,A -85,B 0,C 180,E1 -504.72,E2 -504.72} C_VEL
LIN {X 0,Y 608.453,Z 295.691,A -85,B 0,C 180,E1 -507.477,E2 -507.477} C_VEL
LIN {X 0,Y 608.441,Z 295.693,A -85,B 0,C 180,E1 -510.219,E2 -510.219} C_VEL
LIN {X 0,Y 608.409,Z 295.692,A -85,B 0,C 180,E1 -512.803,E2 -512.803} C_VEL
LIN {X 0,Y 608.436,Z 295.693,A -85,B 0,C 180,E1 -515.428,E2 -515.428} C_VEL
LIN {X 0,Y 608.435,Z 295.692,A -85,B 0,C 180,E1 -518.307,E2 -518.307} C_VEL
LIN {X 0,Y 608.413,Z 295.693,A -85,B 0,C 180,E1 -520.428,E2 -520.428} C_VEL
LIN {X 0,Y 608.422,Z 295.693,A -85,B 0,C 180,E1 -523.215,E2 -523.215} C_VEL
LIN {X 0,Y 608.444,Z 295.695,A -85,B 0,C 180,E1 -525.989,E2 -525.989} C_VEL
LIN {X 0,Y 608.406,Z 295.693,A -85,B 0,C 180,E1 -528.675,E2 -528.675} C_VEL
LIN {X 0,Y 608.442,Z 295.693,A -85,B 0,C 180,E1 -531.364,E2 -531.364} C_VEL
LIN {X 0,Y 608.429,Z 295.695,A -85,B 0,C 180,E1 -534.033,E2 -534.033} C_VEL
LIN {X 0,Y 608.397,Z 295.694,A -85,B 0,C 180,E1 -536.689,E2 -536.689} C_VEL
LIN {X 0,Y 608.465,Z 295.69,A -85,B 0,C 180,E1 -539.338,E2 -539.338} C_VEL
LIN {X 0,Y 608.425,Z 295.696,A -85,B 0,C 180,E1 -541.986,E2 -541.986} C_VEL
LIN {X 0,Y 608.429,Z 295.696,A -85,B 0,C 180,E1 -543.974,E2 -543.974} C_VEL
LIN {X 0,Y 608.423,Z 295.691,A -85,B 0,C 180,E1 -546.633,E2 -546.633} C_VEL
LIN {X 0,Y 608.45,Z 295.692,A -85,B 0,C 180,E1 -549.306,E2 -549.306} C_VEL
LIN {X 0,Y 608.441,Z 295.693,A -85,B 0,C 180,E1 -549.417,E2 -549.417} C_VEL
LIN {X 0,Y 607.757,Z 295.779,A -85,B 0,C 180,E1 -549.97,E2 -549.97} C_VEL
LIN {X 0,Y 604.907,Z 296.132,A -85,B 0,C 180,E1 -550.866,E2 -550.866} C_VEL
LIN {X 0,Y 602.503,Z 296.439,A -85,B 0,C 180,E1 -551.588,E2 -551.588} C_VEL
LIN {X 0,Y 601.46,Z 296.561,A -85,B 0,C 180,E1 -552.144,E2 -552.144} C_VEL
LIN {X 0,Y 601.368,Z 296.57,A -85,B 0,C 180,E1 -552.333,E2 -552.333} C_VEL
LIN {X 0,Y 601.377,Z 296.569,A -85,B 0,C 180,E1 -554.898,E2 -554.898} C_VEL
LIN {X 0,Y 601.374,Z 296.578,A -85,B 0,C 180,E1 -557.689,E2 -557.689} C_VEL
LIN {X 0,Y 601.379,Z 296.574,A -85,B 0,C 180,E1 -559.81,E2 -559.81} C_VEL
LIN {X 0,Y 601.391,Z 296.567,A -85,B 0,C 180,E1 -562.684,E2 -562.684} C_VEL
LIN {X 0,Y 601.425,Z 296.572,A -85,B 0,C 180,E1 -565.618,E2 -565.618} C_VEL
LIN {X 0,Y 601.355,Z 296.575,A -85,B 0,C 180,E1 -567.871,E2 -567.871} C_VEL
LIN {X 0,Y 601.39,Z 296.567,A -85,B 0,C 180,E1 -570.166,E2 -570.166} C_VEL
LIN {X 0,Y 601.382,Z 296.568,A -85,B 0,C 180,E1 -572.711,E2 -572.711} C_VEL
LIN {X 0,Y 601.369,Z 296.574,A -85,B 0,C 180,E1 -575.11,E2 -575.11} C_VEL
LIN {X 0,Y 601.424,Z 296.573,A -85,B 0,C 180,E1 -577.42,E2 -577.42} C_VEL
LIN {X 0,Y 601.37,Z 296.571,A -85,B 0,C 180,E1 -579.999,E2 -579.999} C_VEL
LIN {X 0,Y 601.355,Z 296.572,A -85,B 0,C 180,E1 -582.586,E2 -582.586} C_VEL
LIN {X 0,Y 601.362,Z 296.57,A -85,B 0,C 180,E1 -584.53,E2 -584.53} C_VEL
LIN {X 0,Y 601.377,Z 296.579,A -85,B 0,C 180,E1 -587.413,E2 -587.413} C_VEL
LIN {X 0,Y 601.38,Z 296.57,A -85,B 0,C 180,E1 -590.003,E2 -590.003} C_VEL
LIN {X 0,Y 601.384,Z 296.568,A -85,B 0,C 180,E1 -592.625,E2 -592.625} C_VEL
LIN {X 0,Y 601.41,Z 296.57,A -85,B 0,C 180,E1 -595.069,E2 -595.069} C_VEL
LIN {X 0,Y 601.417,Z 296.572,A -85,B 0,C 180,E1 -597.484,E2 -597.484} C_VEL
LIN {X 0,Y 601.369,Z 296.572,A -85,B 0,C 180,E1 -599.862,E2 -599.862} C_VEL
LIN {X 0,Y 601.356,Z 296.57,A -85,B 0,C 180,E1 -602.13,E2 -602.13} C_VEL
LIN {X 0,Y 601.372,Z 296.569,A -85,B 0,C 180,E1 -604.38,E2 -604.38} C_VEL
LIN {X 0,Y 601.401,Z 296.575,A -85,B 0,C 180,E1 -607.317,E2 -607.317} C_VEL
LIN {X 0,Y 601.414,Z 296.571,A -85,B 0,C 180,E1 -609.478,E2 -609.478} C_VEL
LIN {X 0,Y 601.379,Z 296.571,A -85,B 0,C 180,E1 -611.607,E2 -611.607} C_VEL
LIN {X 0,Y 601.405,Z 296.569,A -85,B 0,C 180,E1 -613.712,E2 -613.712} C_VEL
LIN {X 0,Y 601.425,Z 296.569,A -85,B 0,C 180,E1 -616.829,E2 -616.829} C_VEL
LIN {X 0,Y 601.473,Z 296.881,A -85,B 0,C 180,E1 -617.087,E2 -617.087} C_VEL
LIN {X 0,Y 601.664,Z 298.237,A -85,B 0,C 180,E1 -617.177,E2 -617.177} C_VEL
LIN {X 0,Y 601.63,Z 380.837,A -85,B 0,C 180,E1 -618.183,E2 -618.183} C_VEL
LIN {X 0,Y 601.602,Z 394.145,A -85,B 0,C 180,E1 -618.481,E2 -618.481} C_VEL
LIN {X 0,Y 601.566,Z 407.226,A -85,B 0,C 180,E1 -618.921,E2 -618.921} C_VEL
LIN {X 0,Y 601.514,Z 419.383,A -85,B 0,C 180,E1 -619.481,E2 -619.481} C_VEL
LIN {X 0,Y 601.474,Z 430.804,A -85,B 0,C 180,E1 -620.161,E2 -620.161} C_VEL
LIN {X 0,Y 601.438,Z 441.095,A -85,B 0,C 180,E1 -620.924,E2 -620.924} C_VEL
LIN {X 0,Y 601.411,Z 450.356,A -85,B 0,C 180,E1 -621.77,E2 -621.77} C_VEL
LIN {X 0,Y 601.388,Z 459.329,A -85,B 0,C 180,E1 -622.783,E2 -622.783} C_VEL
LIN {X 0,Y 601.376,Z 466.469,A -85,B 0,C 180,E1 -623.781,E2 -623.781} C_VEL
LIN {X 0,Y 601.373,Z 471.438,A -85,B 0,C 180,E1 -624.636,E2 -624.636} C_VEL
LIN {X 0,Y 601.354,Z 476.181,A -85,B 0,C 180,E1 -625.643,E2 -625.643} C_VEL
LIN {X 0,Y 601.344,Z 479.815,A -85,B 0,C 180,E1 -626.65,E2 -626.65} C_VEL
LIN {X 0,Y 601.324,Z 481.693,A -85,B 0,C 180,E1 -627.32,E2 -627.32} C_VEL
LIN {X 0,Y 601.343,Z 483.127,A -85,B 0,C 180,E1 -627.991,E2 -627.991} C_VEL
LIN {X 0,Y 601.339,Z 484.753,A -85,B 0,C 180,E1 -629.33,E2 -629.33} C_VEL
LIN {X 0,Y 601.336,Z 484.996,A -85,B 0,C 180,E1 -630,E2 -630} C_VEL
LIN {X 0,Y 601.339,Z 484.815,A -85,B 0,C 180,E1 -630.67,E2 -630.67} C_VEL
LIN {X 0,Y 601.343,Z 483.276,A -85,B 0,C 180,E1 -632.009,E2 -632.009} C_VEL
LIN {X 0,Y 601.326,Z 481.917,A -85,B 0,C 180,E1 -632.68,E2 -632.68} C_VEL
LIN {X 0,Y 601.368,Z 479.04,A -85,B 0,C 180,E1 -633.685,E2 -633.685} C_VEL
LIN {X 0,Y 601.337,Z 475.141,A -85,B 0,C 180,E1 -634.693,E2 -634.693} C_VEL
LIN {X 0,Y 601.373,Z 470.11,A -85,B 0,C 180,E1 -635.701,E2 -635.701} C_VEL
LIN {X 0,Y 601.382,Z 463.792,A -85,B 0,C 180,E1 -636.711,E2 -636.711} C_VEL
LIN {X 0,Y 601.396,Z 455.874,A -85,B 0,C 180,E1 -637.723,E2 -637.723} C_VEL
LIN {X 0,Y 601.436,Z 446.031,A -85,B 0,C 180,E1 -638.737,E2 -638.737} C_VEL
LIN {X 0,Y 601.45,Z 435.711,A -85,B 0,C 180,E1 -639.585,E2 -639.585} C_VEL
LIN {X 0,Y 601.498,Z 424.092,A -85,B 0,C 180,E1 -640.349,E2 -640.349} C_VEL
LIN {X 0,Y 601.551,Z 412.85,A -85,B 0,C 180,E1 -640.93,E2 -640.93} C_VEL
LIN {X 0,Y 601.564,Z 400.436,A -85,B 0,C 180,E1 -641.416,E2 -641.416} C_VEL
LIN {X 0,Y 601.602,Z 387.548,A -85,B 0,C 180,E1 -641.775,E2 -641.775} C_VEL
LIN {X 0,Y 601.642,Z 375.267,A -85,B 0,C 180,E1 -641.988,E2 -641.988} C_VEL
LIN {X 0,Y 601.637,Z 297.653,A -85,B 0,C 180,E1 -642.931,E2 -642.931} C_VEL
LIN {X 0,Y 601.417,Z 296.639,A -85,B 0,C 180,E1 -643.064,E2 -643.064} C_VEL
LIN {X 0,Y 601.37,Z 296.571,A -85,B 0,C 180,E1 -645.592,E2 -645.592} C_VEL
LIN {X 0,Y 601.37,Z 296.566,A -85,B 0,C 180,E1 -648.393,E2 -648.393} C_VEL
LIN {X 0,Y 601.382,Z 296.571,A -85,B 0,C 180,E1 -651.24,E2 -651.24} C_VEL
LIN {X 0,Y 601.36,Z 296.572,A -85,B 0,C 180,E1 -653.412,E2 -653.412} C_VEL
LIN {X 0,Y 601.349,Z 296.572,A -85,B 0,C 180,E1 -655.854,E2 -655.854} C_VEL
LIN {X 0,Y 601.414,Z 296.571,A -85,B 0,C 180,E1 -658.627,E2 -658.627} C_VEL
LIN {X 0,Y 601.374,Z 296.569,A -85,B 0,C 180,E1 -661.728,E2 -661.728} C_VEL
LIN {X 0,Y 601.396,Z 296.568,A -85,B 0,C 180,E1 -664.12,E2 -664.12} C_VEL
LIN {X 0,Y 601.387,Z 296.576,A -85,B 0,C 180,E1 -666.583,E2 -666.583} C_VEL
LIN {X 0,Y 601.379,Z 296.569,A -85,B 0,C 180,E1 -669.528,E2 -669.528} C_VEL
LIN {X 0,Y 601.371,Z 296.569,A -85,B 0,C 180,E1 -671.769,E2 -671.769} C_VEL
LIN {X 0,Y 601.394,Z 296.574,A -85,B 0,C 180,E1 -674.532,E2 -674.532} C_VEL
LIN {X 0,Y 601.356,Z 296.572,A -85,B 0,C 180,E1 -677.325,E2 -677.325} C_VEL
LIN {X 0,Y 601.378,Z 296.568,A -85,B 0,C 180,E1 -679.43,E2 -679.43} C_VEL
LIN {X 0,Y 601.345,Z 296.572,A -85,B 0,C 180,E1 -681.726,E2 -681.726} C_VEL
LIN {X 0,Y 601.374,Z 296.569,A -85,B 0,C 180,E1 -683.742,E2 -683.742} C_VEL
LIN {X 0,Y 601.402,Z 296.574,A -85,B 0,C 180,E1 -686.685,E2 -686.685} C_VEL
LIN {X 0,Y 601.382,Z 296.569,A -85,B 0,C 180,E1 -689.056,E2 -689.056} C_VEL
LIN {X 0,Y 601.379,Z 296.567,A -85,B 0,C 180,E1 -691.37,E2 -691.37} C_VEL
LIN {X 0,Y 601.365,Z 296.57,A -85,B 0,C 180,E1 -693.634,E2 -693.634} C_VEL
LIN {X 0,Y 601.387,Z 296.569,A -85,B 0,C 180,E1 -695.857,E2 -695.857} C_VEL
LIN {X 0,Y 601.387,Z 296.573,A -85,B 0,C 180,E1 -698.76,E2 -698.76} C_VEL
LIN {X 0,Y 601.352,Z 296.572,A -85,B 0,C 180,E1 -701.606,E2 -701.606} C_VEL
LIN {X 0,Y 601.38,Z 296.569,A -85,B 0,C 180,E1 -703.711,E2 -703.711} C_VEL
LIN {X 0,Y 601.39,Z 296.577,A -85,B 0,C 180,E1 -706.483,E2 -706.483} C_VEL
LIN {X 0,Y 601.368,Z 296.57,A -85,B 0,C 180,E1 -709.223,E2 -709.223} C_VEL
LIN {X 0,Y 601.39,Z 296.57,A -85,B 0,C 180,E1 -711.938,E2 -711.938} C_VEL
LIN {X 0,Y 601.407,Z 296.571,A -85,B 0,C 180,E1 -714.636,E2 -714.636} C_VEL
LIN {X 0,Y 601.39,Z 296.567,A -85,B 0,C 180,E1 -717.321,E2 -717.321} C_VEL
LIN {X 0,Y 601.415,Z 296.568,A -85,B 0,C 180,E1 -720,E2 -720} C_VEL
LIN {X 0,Y 601.429,Z 296.567,A -85,B 0,C 180,E1 -722.679,E2 -722.679} C_VEL
LIN {X 0,Y 601.376,Z 296.568,A -85,B 0,C 180,E1 -725.365,E2 -725.365} C_VEL
LIN {X 0,Y 601.356,Z 296.571,A -85,B 0,C 180,E1 -727.386,E2 -727.386} C_VEL
LIN {X 0,Y 601.406,Z 296.572,A -85,B 0,C 180,E1 -730.095,E2 -730.095} C_VEL
LIN {X 0,Y 601.393,Z 296.568,A -85,B 0,C 180,E1 -732.829,E2 -732.829} C_VEL
LIN {X 0,Y 601.371,Z 296.571,A -85,B 0,C 180,E1 -735.592,E2 -735.592} C_VEL
LIN {X 0,Y 601.359,Z 296.573,A -85,B 0,C 180,E1 -737.69,E2 -737.69} C_VEL
LIN {X 0,Y 601.417,Z 296.568,A -85,B 0,C 180,E1 -740.522,E2 -740.522} C_VEL
LIN {X 0,Y 601.364,Z 296.571,A -85,B 0,C 180,E1 -743.413,E2 -743.413} C_VEL
LIN {X 0,Y 601.38,Z 296.574,A -85,B 0,C 180,E1 -745.863,E2 -745.863} C_VEL
LIN {X 0,Y 601.409,Z 296.566,A -85,B 0,C 180,E1 -748.786,E2 -748.786} C_VEL
LIN {X 0,Y 601.4,Z 296.567,A -85,B 0,C 180,E1 -751.453,E2 -751.453} C_VEL
LIN {X 0,Y 601.407,Z 296.575,A -85,B 0,C 180,E1 -754.12,E2 -754.12} C_VEL
LIN {X 0,Y 601.37,Z 296.573,A -85,B 0,C 180,E1 -756.585,E2 -756.585} C_VEL
LIN {X 0,Y 601.372,Z 296.569,A -85,B 0,C 180,E1 -759.13,E2 -759.13} C_VEL
LIN {X 0,Y 601.412,Z 296.57,A -85,B 0,C 180,E1 -761.766,E2 -761.766} C_VEL
LIN {X 0,Y 601.393,Z 296.568,A -85,B 0,C 180,E1 -764.533,E2 -764.533} C_VEL
LIN {X 0,Y 601.355,Z 296.572,A -85,B 0,C 180,E1 -767.326,E2 -767.326} C_VEL
LIN {X 0,Y 601.395,Z 296.577,A -85,B 0,C 180,E1 -770.005,E2 -770.005} C_VEL
LIN {X 0,Y 601.391,Z 296.569,A -85,B 0,C 180,E1 -772.624,E2 -772.624} C_VEL
LIN {X 0,Y 601.365,Z 296.57,A -85,B 0,C 180,E1 -775.065,E2 -775.065} C_VEL
LIN {X 0,Y 601.399,Z 296.569,A -85,B 0,C 180,E1 -777.483,E2 -777.483} C_VEL
LIN {X 0,Y 601.406,Z 296.574,A -85,B 0,C 180,E1 -779.856,E2 -779.856} C_VEL
LIN {X 0,Y 601.373,Z 296.575,A -85,B 0,C 180,E1 -782.886,E2 -782.886} C_VEL
LIN {X 0,Y 601.406,Z 296.744,A -85,B 0,C 180,E1 -783.614,E2 -783.614} C_VEL
LIN {X 0,Y 601.984,Z 299.994,A -85,B 0,C 180,E1 -784.021,E2 -784.021} C_VEL
LIN {X 0,Y 601.83,Z 325.517,A -85,B 0,C 180,E1 -786.807,E2 -786.807} C_VEL
LIN {X 0,Y 601.739,Z 350.563,A -85,B 0,C 180,E1 -789.49,E2 -789.49} C_VEL
LIN {X 0,Y 601.624,Z 377.459,A -85,B 0,C 180,E1 -792.319,E2 -792.319} C_VEL
LIN {X 0,Y 601.543,Z 404.355,A -85,B 0,C 180,E1 -795.106,E2 -795.106} C_VEL
LIN {X 0,Y 601.517,Z 420.904,A -85,B 0,C 180,E1 -796.788,E2 -796.788} C_VEL
LIN {X 0,Y 601.668,Z 426.739,A -85,B 0,C 180,E1 -796.877,E2 -796.877} C_VEL
LIN {X 0,Y 601.605,Z 530.958,A -85,B 0,C 180,E1 -798.14,E2 -798.14} C_VEL
LIN {X 0,Y 601.587,Z 544.224,A -85,B 0,C 180,E1 -798.438,E2 -798.438} C_VEL
LIN {X 0,Y 601.549,Z 555.926,A -85,B 0,C 180,E1 -798.826,E2 -798.826} C_VEL
LIN {X 0,Y 601.517,Z 566.927,A -85,B 0,C 180,E1 -799.311,E2 -799.311} C_VEL
LIN {X 0,Y 601.479,Z 577.583,A -85,B 0,C 180,E1 -799.906,E2 -799.906} C_VEL
LIN {X 0,Y 601.446,Z 588.478,A -85,B 0,C 180,E1 -800.67,E2 -800.67} C_VEL
LIN {X 0,Y 601.429,Z 599.113,A -85,B 0,C 180,E1 -801.601,E2 -801.601} C_VEL
LIN {X 0,Y 601.418,Z 606.961,A -85,B 0,C 180,E1 -802.446,E2 -802.446} C_VEL
LIN {X 0,Y 601.37,Z 614.225,A -85,B 0,C 180,E1 -803.398,E2 -803.398} C_VEL
LIN {X 0,Y 601.372,Z 619.867,A -85,B 0,C 180,E1 -804.299,E2 -804.299} C_VEL
LIN {X 0,Y 601.337,Z 624.95,A -85,B 0,C 180,E1 -805.307,E2 -805.307} C_VEL
LIN {X 0,Y 601.367,Z 628.896,A -85,B 0,C 180,E1 -806.315,E2 -806.315} C_VEL
LIN {X 0,Y 601.325,Z 631.809,A -85,B 0,C 180,E1 -807.32,E2 -807.32} C_VEL
LIN {X 0,Y 601.341,Z 633.202,A -85,B 0,C 180,E1 -807.991,E2 -807.991} C_VEL
LIN {X 0,Y 601.339,Z 634.784,A -85,B 0,C 180,E1 -809.33,E2 -809.33} C_VEL
LIN {X 0,Y 601.335,Z 635,A -85,B 0,C 180,E1 -810,E2 -810} C_VEL
LIN {X 0,Y 601.348,Z 634.184,A -85,B 0,C 180,E1 -811.339,E2 -811.339} C_VEL
LIN {X 0,Y 601.341,Z 633.202,A -85,B 0,C 180,E1 -812.009,E2 -812.009} C_VEL
LIN {X 0,Y 601.325,Z 631.809,A -85,B 0,C 180,E1 -812.68,E2 -812.68} C_VEL
LIN {X 0,Y 601.367,Z 628.896,A -85,B 0,C 180,E1 -813.685,E2 -813.685} C_VEL
LIN {X 0,Y 601.337,Z 624.95,A -85,B 0,C 180,E1 -814.693,E2 -814.693} C_VEL
LIN {X 0,Y 601.372,Z 618.878,A -85,B 0,C 180,E1 -815.869,E2 -815.869} C_VEL
LIN {X 0,Y 601.382,Z 612.236,A -85,B 0,C 180,E1 -816.88,E2 -816.88} C_VEL
LIN {X 0,Y 601.4,Z 603.991,A -85,B 0,C 180,E1 -817.892,E2 -817.892} C_VEL
LIN {X 0,Y 601.436,Z 595.539,A -85,B 0,C 180,E1 -818.737,E2 -818.737} C_VEL
LIN {X 0,Y 601.442,Z 585.095,A -85,B 0,C 180,E1 -819.585,E2 -819.585} C_VEL
LIN {X 0,Y 601.473,Z 574.76,A -85,B 0,C 180,E1 -820.264,E2 -820.264} C_VEL
LIN {X 0,Y 601.537,Z 563.898,A -85,B 0,C 180,E1 -820.836,E2 -820.836} C_VEL
LIN {X 0,Y 601.565,Z 551.378,A -85,B 0,C 180,E1 -821.34,E2 -821.34} C_VEL
LIN {X 0,Y 601.598,Z 538.361,A -85,B 0,C 180,E1 -821.711,E2 -821.711} C_VEL
LIN {X 0,Y 601.614,Z 525.101,A -85,B 0,C 180,E1 -821.946,E2 -821.946} C_VEL
LIN {X 0,Y 601.575,Z 421.549,A -85,B 0,C 180,E1 -823.19,E2 -823.19} C_VEL
LIN {X 0,Y 601.517,Z 420.348,A -85,B 0,C 180,E1 -823.255,E2 -823.255} C_VEL
LIN {X 0,Y 601.589,Z 392.588,A -85,B 0,C 180,E1 -826.108,E2 -826.108} C_VEL
LIN {X 0,Y 601.69,Z 364.011,A -85,B 0,C 180,E1 -829.09,E2 -829.09} C_VEL
LIN {X 0,Y 601.775,Z 338.797,A -85,B 0,C 180,E1 -831.765,E2 -831.765} C_VEL
LIN {X 0,Y 601.891,Z 314.504,A -85,B 0,C 180,E1 -834.388,E2 -834.388} C_VEL
LIN {X 0,Y 601.957,Z 299.013,A -85,B 0,C 180,E1 -836.089,E2 -836.089} C_VEL
LIN {X 0,Y 601.416,Z 296.663,A -85,B 0,C 180,E1 -836.409,E2 -836.409} C_VEL
LIN {X 0,Y 601.392,Z 296.568,A -85,B 0,C 180,E1 -839.394,E2 -839.394} C_VEL
LIN {X 0,Y 601.388,Z 296.573,A -85,B 0,C 180,E1 -841.727,E2 -841.727} C_VEL
LIN {X 0,Y 601.406,Z 296.574,A -85,B 0,C 180,E1 -844.119,E2 -844.119} C_VEL
LIN {X 0,Y 601.37,Z 296.572,A -85,B 0,C 180,E1 -846.585,E2 -846.585} C_VEL
LIN {X 0,Y 601.378,Z 296.568,A -85,B 0,C 180,E1 -849.128,E2 -849.128} C_VEL
LIN {X 0,Y 601.411,Z 296.571,A -85,B 0,C 180,E1 -851.765,E2 -851.765} C_VEL
LIN {X 0,Y 601.393,Z 296.567,A -85,B 0,C 180,E1 -854.532,E2 -854.532} C_VEL
LIN {X 0,Y 601.381,Z 296.57,A -85,B 0,C 180,E1 -857.411,E2 -857.411} C_VEL
LIN {X 0,Y 601.389,Z 296.576,A -85,B 0,C 180,E1 -860.003,E2 -860.003} C_VEL
LIN {X 0,Y 601.384,Z 296.566,A -85,B 0,C 180,E1 -862.623,E2 -862.623} C_VEL
LIN {X 0,Y 601.37,Z 296.569,A -85,B 0,C 180,E1 -865.065,E2 -865.065} C_VEL
LIN {X 0,Y 601.422,Z 296.567,A -85,B 0,C 180,E1 -867.484,E2 -867.484} C_VEL
LIN {X 0,Y 601.443,Z 296.571,A -85,B 0,C 180,E1 -869.847,E2 -869.847} C_VEL
LIN {X 0,Y 601.365,Z 296.57,A -85,B 0,C 180,E1 -872.645,E2 -872.645} C_VEL
LIN {X 0,Y 601.429,Z 296.571,A -85,B 0,C 180,E1 -875.707,E2 -875.707} C_VEL
LIN {X 0,Y 601.393,Z 296.573,A -85,B 0,C 180,E1 -878.04,E2 -878.04} C_VEL
LIN {X 0,Y 601.379,Z 296.572,A -85,B 0,C 180,E1 -880.19,E2 -880.19} C_VEL
LIN {X 0,Y 601.391,Z 296.567,A -85,B 0,C 180,E1 -883.013,E2 -883.013} C_VEL
LIN {X 0,Y 601.391,Z 296.575,A -85,B 0,C 180,E1 -885.916,E2 -885.916} C_VEL
LIN {X 0,Y 601.387,Z 296.568,A -85,B 0,C 180,E1 -888.541,E2 -888.541} C_VEL
LIN {X 0,Y 601.397,Z 296.569,A -85,B 0,C 180,E1 -891.262,E2 -891.262} C_VEL
LIN {X 0,Y 601.385,Z 296.574,A -85,B 0,C 180,E1 -893.963,E2 -893.963} C_VEL
LIN {X 0,Y 601.378,Z 296.575,A -85,B 0,C 180,E1 -895.979,E2 -895.979} C_VEL
LIN {X 0,Y 601.398,Z 296.571,A -85,B 0,C 180,E1 -897.991,E2 -897.991} C_VEL
LIN {X 0,Y 601.42,Z 296.568,A -85,B 0,C 180,E1 -900,E2 -900} C_VEL
LIN {X 0,Y 601.391,Z 296.567,A -85,B 0,C 180,E1 -902.679,E2 -902.679} C_VEL
LIN {X 0,Y 601.41,Z 296.57,A -85,B 0,C 180,E1 -905.364,E2 -905.364} C_VEL
LIN {X 0,Y 601.416,Z 296.567,A -85,B 0,C 180,E1 -908.061,E2 -908.061} C_VEL
LIN {X 0,Y 601.391,Z 296.568,A -85,B 0,C 180,E1 -911,E2 -911} C_VEL
LIN {X 0,Y 601.368,Z 296.57,A -85,B 0,C 180,E1 -912.333,E2 -912.333} C_VEL
LIN {X 0,Y 600.686,Z 296.656,A -85,B 0,C 180,E1 -912.892,E2 -912.892} C_VEL
LIN {X 0,Y 597.836,Z 297.016,A -85,B 0,C 180,E1 -913.8,E2 -913.8} C_VEL
LIN {X 0,Y 595.438,Z 297.312,A -85,B 0,C 180,E1 -914.53,E2 -914.53} C_VEL
LIN {X 0,Y 594.409,Z 297.438,A -85,B 0,C 180,E1 -915.094,E2 -915.094} C_VEL
LIN {X 0,Y 594.325,Z 297.449,A -85,B 0,C 180,E1 -915.284,E2 -915.284} C_VEL
LIN {X 0,Y 594.32,Z 297.453,A -85,B 0,C 180,E1 -917.906,E2 -917.906} C_VEL
LIN {X 0,Y 594.367,Z 297.442,A -85,B 0,C 180,E1 -920.777,E2 -920.777} C_VEL
LIN {X 0,Y 594.339,Z 297.453,A -85,B 0,C 180,E1 -923.706,E2 -923.706} C_VEL
LIN {X 0,Y 594.345,Z 297.447,A -85,B 0,C 180,E1 -926.017,E2 -926.017} C_VEL
LIN {X 0,Y 594.361,Z 297.443,A -85,B 0,C 180,E1 -929,E2 -929} C_VEL
LIN {X 0,Y 594.361,Z 297.45,A -85,B 0,C 180,E1 -931.642,E2 -931.642} C_VEL
LIN {X 0,Y 594.35,Z 297.445,A -85,B 0,C 180,E1 -934.136,E2 -934.136} C_VEL
LIN {X 0,Y 594.368,Z 297.446,A -85,B 0,C 180,E1 -937.088,E2 -937.088} C_VEL
LIN {X 0,Y 594.332,Z 297.45,A -85,B 0,C 180,E1 -939.77,E2 -939.77} C_VEL
LIN {X 0,Y 594.323,Z 297.447,A -85,B 0,C 180,E1 -942.38,E2 -942.38} C_VEL
LIN {X 0,Y 594.31,Z 297.451,A -85,B 0,C 180,E1 -944.805,E2 -944.805} C_VEL
LIN {X 0,Y 594.338,Z 297.452,A -85,B 0,C 180,E1 -947.623,E2 -947.623} C_VEL
LIN {X 0,Y 594.347,Z 297.445,A -85,B 0,C 180,E1 -950.318,E2 -950.318} C_VEL
LIN {X 0,Y 594.348,Z 297.447,A -85,B 0,C 180,E1 -952.911,E2 -952.911} C_VEL
LIN {X 0,Y 594.353,Z 297.446,A -85,B 0,C 180,E1 -955.866,E2 -955.866} C_VEL
LIN {X 0,Y 594.338,Z 297.446,A -85,B 0,C 180,E1 -958.649,E2 -958.649} C_VEL
LIN {X 0,Y 594.374,Z 297.447,A -85,B 0,C 180,E1 -961.044,E2 -961.044} C_VEL
LIN {X 0,Y 594.338,Z 297.446,A -85,B 0,C 180,E1 -964.055,E2 -964.055} C_VEL
LIN {X 0,Y 594.343,Z 297.451,A -85,B 0,C 180,E1 -967.032,E2 -967.032} C_VEL
LIN {X 0,Y 594.347,Z 297.446,A -85,B 0,C 180,E1 -969.946,E2 -969.946} C_VEL
LIN {X 0,Y 594.318,Z 297.444,A -85,B 0,C 180,E1 -972.094,E2 -972.094} C_VEL
LIN {X 0,Y 594.33,Z 297.448,A -85,B 0,C 180,E1 -974.218,E2 -974.218} C_VEL
LIN {X 0,Y 594.435,Z 297.594,A -85,B 0,C 180,E1 -976.91,E2 -976.91} C_VEL
LIN {X 0,Y 594.64,Z 298.703,A -85,B 0,C 180,E1 -977.023,E2 -977.023} C_VEL
LIN {X 0,Y 594.686,Z 380.867,A -85,B 0,C 180,E1 -978.043,E2 -978.043} C_VEL
LIN {X 0,Y 594.636,Z 394.166,A -85,B 0,C 180,E1 -978.344,E2 -978.344} C_VEL
LIN {X 0,Y 594.595,Z 406.159,A -85,B 0,C 180,E1 -978.748,E2 -978.748} C_VEL
LIN {X 0,Y 594.553,Z 417.768,A -85,B 0,C 180,E1 -979.271,E2 -979.271} C_VEL
LIN {X 0,Y 594.486,Z 429.534,A -85,B 0,C 180,E1 -979.958,E2 -979.958} C_VEL
LIN {X 0,Y 594.414,Z 440.044,A -85,B 0,C 180,E1 -980.73,E2 -980.73} C_VEL
LIN {X 0,Y 594.384,Z 448.648,A -85,B 0,C 180,E1 -981.501,E2 -981.501} C_VEL
LIN {X 0,Y 594.347,Z 456.574,A -85,B 0,C 180,E1 -982.356,E2 -982.356} C_VEL
LIN {X 0,Y 594.305,Z 464.395,A -85,B 0,C 180,E1 -983.39,E2 -983.39} C_VEL
LIN {X 0,Y 594.289,Z 471.441,A -85,B 0,C 180,E1 -984.571,E2 -984.571} C_VEL
LIN {X 0,Y 594.27,Z 476.184,A -85,B 0,C 180,E1 -985.591,E2 -985.591} C_VEL
LIN {X 0,Y 594.267,Z 479.817,A -85,B 0,C 180,E1 -986.61,E2 -986.61} C_VEL
LIN {X 0,Y 594.225,Z 481.695,A -85,B 0,C 180,E1 -987.288,E2 -987.288} C_VEL
LIN {X 0,Y 594.242,Z 483.127,A -85,B 0,C 180,E1 -987.967,E2 -987.967} C_VEL
LIN {X 0,Y 594.24,Z 484.753,A -85,B 0,C 180,E1 -989.322,E2 -989.322} C_VEL
LIN {X 0,Y 594.236,Z 484.996,A -85,B 0,C 180,E1 -990,E2 -990} C_VEL
LIN {X 0,Y 594.239,Z 484.815,A -85,B 0,C 180,E1 -990.678,E2 -990.678} C_VEL
LIN {X 0,Y 594.242,Z 483.276,A -85,B 0,C 180,E1 -992.033,E2 -992.033} C_VEL
LIN {X 0,Y 594.226,Z 481.915,A -85,B 0,C 180,E1 -992.712,E2 -992.712} C_VEL
LIN {X 0,Y 594.289,Z 479.038,A -85,B 0,C 180,E1 -993.729,E2 -993.729} C_VEL
LIN {X 0,Y 594.242,Z 475.139,A -85,B 0,C 180,E1 -994.749,E2 -994.749} C_VEL
LIN {X 0,Y 594.299,Z 470.108,A -85,B 0,C 180,E1 -995.769,E2 -995.769} C_VEL
LIN {X 0,Y 594.316,Z 463.788,A -85,B 0,C 180,E1 -996.791,E2 -996.791} C_VEL
LIN {X 0,Y 594.346,Z 455.869,A -85,B 0,C 180,E1 -997.815,E2 -997.815} C_VEL
LIN {X 0,Y 594.381,Z 446.024,A -85,B 0,C 180,E1 -998.842,E2 -998.842} C_VEL
LIN {X 0,Y 594.433,Z 435.706,A -85,B 0,C 180,E1 -999.699,E2 -999.699} C_VEL
LIN {X 0,Y 594.516,Z 424.08,A -85,B 0,C 180,E1 -1000.472,E2 -1000.472} C_VEL
LIN {X 0,Y 594.541,Z 412.257,A -85,B 0,C 180,E1 -1001.086,E2 -1001.086} C_VEL
LIN {X 0,Y 594.612,Z 399.24,A -85,B 0,C 180,E1 -1001.591,E2 -1001.591} C_VEL
LIN {X 0,Y 594.668,Z 386.607,A -85,B 0,C 180,E1 -1001.936,E2 -1001.936} C_VEL
LIN {X 0,Y 594.702,Z 373.469,A -85,B 0,C 180,E1 -1002.152,E2 -1002.152} C_VEL
LIN {X 0,Y 594.679,Z 298.787,A -85,B 0,C 180,E1 -1003.063,E2 -1003.063} C_VEL
LIN {X 0,Y 594.395,Z 297.612,A -85,B 0,C 180,E1 -1003.178,E2 -1003.178} C_VEL
LIN {X 0,Y 594.324,Z 297.448,A -85,B 0,C 180,E1 -1005.782,E2 -1005.782} C_VEL
LIN {X 0,Y 594.369,Z 297.451,A -85,B 0,C 180,E1 -1008.924,E2 -1008.924} C_VEL
LIN {X 0,Y 594.338,Z 297.446,A -85,B 0,C 180,E1 -1011.504,E2 -1011.504} C_VEL
LIN {X 0,Y 594.329,Z 297.447,A -85,B 0,C 180,E1 -1013.706,E2 -1013.706} C_VEL
LIN {X 0,Y 594.346,Z 297.454,A -85,B 0,C 180,E1 -1016.701,E2 -1016.701} C_VEL
LIN {X 0,Y 594.368,Z 297.448,A -85,B 0,C 180,E1 -1018.999,E2 -1018.999} C_VEL
LIN {X 0,Y 594.349,Z 297.444,A -85,B 0,C 180,E1 -1021.638,E2 -1021.638} C_VEL
LIN {X 0,Y 594.369,Z 297.45,A -85,B 0,C 180,E1 -1024.58,E2 -1024.58} C_VEL
LIN {X 0,Y 594.345,Z 297.444,A -85,B 0,C 180,E1 -1027.602,E2 -1027.602} C_VEL
LIN {X 0,Y 594.349,Z 297.453,A -85,B 0,C 180,E1 -1030.568,E2 -1030.568} C_VEL
LIN {X 0,Y 594.335,Z 297.446,A -85,B 0,C 180,E1 -1033.301,E2 -1033.301} C_VEL
LIN {X 0,Y 594.329,Z 297.45,A -85,B 0,C 180,E1 -1036.163,E2 -1036.163} C_VEL
LIN {X 0,Y 594.353,Z 297.445,A -85,B 0,C 180,E1 -1039.18,E2 -1039.18} C_VEL
LIN {X 0,Y 594.34,Z 297.446,A -85,B 0,C 180,E1 -1042.056,E2 -1042.056} C_VEL
LIN {X 0,Y 594.312,Z 297.458,A -85,B 0,C 180,E1 -1044.68,E2 -1044.68} C_VEL
LIN {X 0,Y 594.361,Z 297.445,A -85,B 0,C 180,E1 -1047.09,E2 -1047.09} C_VEL
LIN {X 0,Y 594.339,Z 297.443,A -85,B 0,C 180,E1 -1049.678,E2 -1049.678} C_VEL
LIN {X 0,Y 594.306,Z 297.448,A -85,B 0,C 180,E1 -1051.769,E2 -1051.769} C_VEL
LIN {X 0,Y 594.348,Z 297.447,A -85,B 0,C 180,E1 -1054.054,E2 -1054.054} C_VEL
LIN {X 0,Y 594.317,Z 297.45,A -85,B 0,C 180,E1 -1057.031,E2 -1057.031} C_VEL
LIN {X 0,Y 594.364,Z 297.442,A -85,B 0,C 180,E1 -1059.223,E2 -1059.223} C_VEL
LIN {X 0,Y 594.317,Z 297.452,A -85,B 0,C 180,E1 -1062.094,E2 -1062.094} C_VEL
LIN {X 0,Y 594.33,Z 297.449,A -85,B 0,C 180,E1 -1064.921,E2 -1064.921} C_VEL
LIN {X 0,Y 594.333,Z 297.447,A -85,B 0,C 180,E1 -1067.71,E2 -1067.71} C_VEL
LIN {X 0,Y 594.34,Z 297.454,A -85,B 0,C 180,E1 -1070.471,E2 -1070.471} C_VEL
LIN {X 0,Y 594.325,Z 297.447,A -85,B 0,C 180,E1 -1073.362,E2 -1073.362} C_VEL
LIN {X 0,Y 594.325,Z 297.451,A -85,B 0,C 180,E1 -1075.931,E2 -1075.931} C_VEL
LIN {X 0,Y 594.363,Z 297.447,A -85,B 0,C 180,E1 -1078.645,E2 -1078.645} C_VEL
LIN {X 0,Y 594.408,Z 297.442,A -85,B 0,C 180,E1 -1080.677,E2 -1080.677} C_VEL
LIN {X 0,Y 594.303,Z 297.45,A -85,B 0,C 180,E1 -1083.39,E2 -1083.39} C_VEL
LIN {X 0,Y 594.344,Z 297.444,A -85,B 0,C 180,E1 -1085.428,E2 -1085.428} C_VEL
LIN {X 0,Y 594.33,Z 297.446,A -85,B 0,C 180,E1 -1087.474,E2 -1087.474} C_VEL
LIN {X 0,Y 594.366,Z 297.452,A -85,B 0,C 180,E1 -1090.216,E2 -1090.216} C_VEL
LIN {X 0,Y 594.336,Z 297.446,A -85,B 0,C 180,E1 -1092.984,E2 -1092.984} C_VEL
LIN {X 0,Y 594.345,Z 297.445,A -85,B 0,C 180,E1 -1095.079,E2 -1095.079} C_VEL
LIN {X 0,Y 594.329,Z 297.447,A -85,B 0,C 180,E1 -1097.195,E2 -1097.195} C_VEL
LIN {X 0,Y 594.353,Z 297.45,A -85,B 0,C 180,E1 -1100.055,E2 -1100.055} C_VEL
LIN {X 0,Y 594.339,Z 297.446,A -85,B 0,C 180,E1 -1102.968,E2 -1102.968} C_VEL
LIN {X 0,Y 594.315,Z 297.448,A -85,B 0,C 180,E1 -1105.196,E2 -1105.196} C_VEL
LIN {X 0,Y 594.334,Z 297.447,A -85,B 0,C 180,E1 -1107.519,E2 -1107.519} C_VEL
LIN {X 0,Y 594.378,Z 297.448,A -85,B 0,C 180,E1 -1110.328,E2 -1110.328} C_VEL
LIN {X 0,Y 594.367,Z 297.442,A -85,B 0,C 180,E1 -1112.951,E2 -1112.951} C_VEL
LIN {X 0,Y 594.308,Z 297.45,A -85,B 0,C 180,E1 -1115.412,E2 -1115.412} C_VEL
LIN {X 0,Y 594.364,Z 297.45,A -85,B 0,C 180,E1 -1117.943,E2 -1117.943} C_VEL
LIN {X 0,Y 594.35,Z 297.445,A -85,B 0,C 180,E1 -1120.82,E2 -1120.82} C_VEL
LIN {X 0,Y 594.337,Z 297.446,A -85,B 0,C 180,E1 -1123.302,E2 -1123.302} C_VEL
LIN {X 0,Y 594.34,Z 297.454,A -85,B 0,C 180,E1 -1126.164,E2 -1126.164} C_VEL
LIN {X 0,Y 594.361,Z 297.445,A -85,B 0,C 180,E1 -1128.535,E2 -1128.535} C_VEL
LIN {X 0,Y 594.358,Z 297.443,A -85,B 0,C 180,E1 -1131.299,E2 -1131.299} C_VEL
LIN {X 0,Y 594.34,Z 297.452,A -85,B 0,C 180,E1 -1133.755,E2 -1133.755} C_VEL
LIN {X 0,Y 594.35,Z 297.45,A -85,B 0,C 180,E1 -1136.238,E2 -1136.238} C_VEL
LIN {X 0,Y 594.354,Z 297.445,A -85,B 0,C 180,E1 -1138.649,E2 -1138.649} C_VEL
LIN {X 0,Y 594.335,Z 297.446,A -85,B 0,C 180,E1 -1141.051,E2 -1141.051} C_VEL
LIN {X 0,Y 594.37,Z 297.672,A -85,B 0,C 180,E1 -1143.387,E2 -1143.387} C_VEL
LIN {X 0,Y 595.233,Z 302.361,A -85,B 0,C 180,E1 -1143.97,E2 -1143.97} C_VEL
LIN {X 0,Y 595.027,Z 327.03,A -85,B 0,C 180,E1 -1146.692,E2 -1146.692} C_VEL
LIN {X 0,Y 594.832,Z 353.925,A -85,B 0,C 180,E1 -1149.602,E2 -1149.602} C_VEL
LIN {X 0,Y 594.678,Z 379.14,A -85,B 0,C 180,E1 -1152.283,E2 -1152.283} C_VEL
LIN {X 0,Y 594.565,Z 406.036,A -85,B 0,C 180,E1 -1155.103,E2 -1155.103} C_VEL
LIN {X 0,Y 594.553,Z 421.131,A -85,B 0,C 180,E1 -1156.641,E2 -1156.641} C_VEL
LIN {X 0,Y 594.755,Z 426.739,A -85,B 0,C 180,E1 -1156.722,E2 -1156.722} C_VEL
LIN {X 0,Y 594.684,Z 530.958,A -85,B 0,C 180,E1 -1158,E2 -1158} C_VEL
LIN {X 0,Y 594.64,Z 543.465,A -85,B 0,C 180,E1 -1158.28,E2 -1158.28} C_VEL
LIN {X 0,Y 594.595,Z 556.577,A -85,B 0,C 180,E1 -1158.719,E2 -1158.719} C_VEL
LIN {X 0,Y 594.539,Z 568.636,A -85,B 0,C 180,E1 -1159.27,E2 -1159.27} C_VEL
LIN {X 0,Y 594.469,Z 580.203,A -85,B 0,C 180,E1 -1159.958,E2 -1159.958} C_VEL
LIN {X 0,Y 594.413,Z 590.598,A -85,B 0,C 180,E1 -1160.73,E2 -1160.73} C_VEL
LIN {X 0,Y 594.383,Z 599.114,A -85,B 0,C 180,E1 -1161.501,E2 -1161.501} C_VEL
LIN {X 0,Y 594.347,Z 606.961,A -85,B 0,C 180,E1 -1162.356,E2 -1162.356} C_VEL
LIN {X 0,Y 594.282,Z 614.813,A -85,B 0,C 180,E1 -1163.408,E2 -1163.408} C_VEL
LIN {X 0,Y 594.289,Z 621.681,A -85,B 0,C 180,E1 -1164.571,E2 -1164.571} C_VEL
LIN {X 0,Y 594.27,Z 626.372,A -85,B 0,C 180,E1 -1165.591,E2 -1165.591} C_VEL
LIN {X 0,Y 594.267,Z 629.956,A -85,B 0,C 180,E1 -1166.61,E2 -1166.61} C_VEL
LIN {X 0,Y 594.226,Z 631.809,A -85,B 0,C 180,E1 -1167.288,E2 -1167.288} C_VEL
LIN {X 0,Y 594.24,Z 633.201,A -85,B 0,C 180,E1 -1167.967,E2 -1167.967} C_VEL
LIN {X 0,Y 594.239,Z 634.784,A -85,B 0,C 180,E1 -1169.322,E2 -1169.322} C_VEL
LIN {X 0,Y 594.236,Z 635,A -85,B 0,C 180,E1 -1170,E2 -1170} C_VEL
LIN {X 0,Y 594.247,Z 634.185,A -85,B 0,C 180,E1 -1171.355,E2 -1171.355} C_VEL
LIN {X 0,Y 594.24,Z 633.202,A -85,B 0,C 180,E1 -1172.033,E2 -1172.033} C_VEL
LIN {X 0,Y 594.226,Z 631.81,A -85,B 0,C 180,E1 -1172.712,E2 -1172.712} C_VEL
LIN {X 0,Y 594.288,Z 628.896,A -85,B 0,C 180,E1 -1173.729,E2 -1173.729} C_VEL
LIN {X 0,Y 594.242,Z 624.95,A -85,B 0,C 180,E1 -1174.749,E2 -1174.749} C_VEL
LIN {X 0,Y 594.304,Z 618.878,A -85,B 0,C 180,E1 -1175.939,E2 -1175.939} C_VEL
LIN {X 0,Y 594.308,Z 612.237,A -85,B 0,C 180,E1 -1176.962,E2 -1176.962} C_VEL
LIN {X 0,Y 594.359,Z 603.991,A -85,B 0,C 180,E1 -1177.986,E2 -1177.986} C_VEL
LIN {X 0,Y 594.382,Z 595.539,A -85,B 0,C 180,E1 -1178.842,E2 -1178.842} C_VEL
LIN {X 0,Y 594.427,Z 585.096,A -85,B 0,C 180,E1 -1179.699,E2 -1179.699} C_VEL
LIN {X 0,Y 594.486,Z 574.762,A -85,B 0,C 180,E1 -1180.386,E2 -1180.386} C_VEL
LIN {X 0,Y 594.561,Z 563.691,A -85,B 0,C 180,E1 -1180.975,E2 -1180.975} C_VEL
LIN {X 0,Y 594.6,Z 551.706,A -85,B 0,C 180,E1 -1181.464,E2 -1181.464} C_VEL
LIN {X 0,Y 594.643,Z 538.36,A -85,B 0,C 180,E1 -1181.85,E2 -1181.85} C_VEL
LIN {X 0,Y 594.691,Z 525.101,A -85,B 0,C 180,E1 -1182.087,E2 -1182.087} C_VEL
LIN {X 0,Y 594.604,Z 421.535,A -85,B 0,C 180,E1 -1183.347,E2 -1183.347} C_VEL
LIN {X 0,Y 594.48,Z 420.348,A -85,B 0,C 180,E1 -1183.415,E2 -1183.415} C_VEL
LIN {X 0,Y 594.635,Z 392.588,A -85,B 0,C 180,E1 -1186.302,E2 -1186.302} C_VEL
LIN {X 0,Y 594.765,Z 364.011,A -85,B 0,C 180,E1 -1189.321,E2 -1189.321} C_VEL
LIN {X 0,Y 594.937,Z 338.797,A -85,B 0,C 180,E1 -1192.028,E2 -1192.028} C_VEL
LIN {X 0,Y 595.157,Z 313.432,A -85,B 0,C 180,E1 -1194.801,E2 -1194.801} C_VEL
LIN {X 0,Y 595.222,Z 300.972,A -85,B 0,C 180,E1 -1196.187,E2 -1196.187} C_VEL
LIN {X 0,Y 594.366,Z 297.567,A -85,B 0,C 180,E1 -1196.641,E2 -1196.641} C_VEL
LIN {X 0,Y 594.335,Z 297.446,A -85,B 0,C 180,E1 -1199,E2 -1199} C_VEL
LIN {X 0,Y 594.366,Z 297.446,A -85,B 0,C 180,E1 -1201.64,E2 -1201.64} C_VEL
LIN {X 0,Y 594.349,Z 297.446,A -85,B 0,C 180,E1 -1204.581,E2 -1204.581} C_VEL
LIN {X 0,Y 594.358,Z 297.447,A -85,B 0,C 180,E1 -1207.604,E2 -1207.604} C_VEL
LIN {X 0,Y 594.347,Z 297.446,A -85,B 0,C 180,E1 -1210.568,E2 -1210.568} C_VEL
LIN {X 0,Y 594.334,Z 297.447,A -85,B 0,C 180,E1 -1213.301,E2 -1213.301} C_VEL
LIN {X 0,Y 594.338,Z 297.452,A -85,B 0,C 180,E1 -1216.162,E2 -1216.162} C_VEL
LIN {X 0,Y 594.357,Z 297.445,A -85,B 0,C 180,E1 -1218.534,E2 -1218.534} C_VEL
LIN {X 0,Y 594.358,Z 297.443,A -85,B 0,C 180,E1 -1221.298,E2 -1221.298} C_VEL
LIN {X 0,Y 594.338,Z 297.45,A -85,B 0,C 180,E1 -1223.754,E2 -1223.754} C_VEL
LIN {X 0,Y 594.353,Z 297.448,A -85,B 0,C 180,E1 -1226.237,E2 -1226.237} C_VEL
LIN {X 0,Y 594.35,Z 297.445,A -85,B 0,C 180,E1 -1228.648,E2 -1228.648} C_VEL
LIN {X 0,Y 594.367,Z 297.441,A -85,B 0,C 180,E1 -1231.043,E2 -1231.043} C_VEL
LIN {X 0,Y 594.347,Z 297.451,A -85,B 0,C 180,E1 -1234.054,E2 -1234.054} C_VEL
LIN {X 0,Y 594.358,Z 297.446,A -85,B 0,C 180,E1 -1236.295,E2 -1236.295} C_VEL
LIN {X 0,Y 594.388,Z 297.439,A -85,B 0,C 180,E1 -1239.224,E2 -1239.224} C_VEL
LIN {X 0,Y 594.323,Z 297.453,A -85,B 0,C 180,E1 -1242.094,E2 -1242.094} C_VEL
LIN {X 0,Y 594.337,Z 297.449,A -85,B 0,C 180,E1 -1244.218,E2 -1244.218} C_VEL
LIN {X 0,Y 594.345,Z 297.446,A -85,B 0,C 180,E1 -1246.32,E2 -1246.32} C_VEL
LIN {X 0,Y 594.343,Z 297.446,A -85,B 0,C 180,E1 -1249.094,E2 -1249.094} C_VEL
LIN {X 0,Y 594.348,Z 297.453,A -85,B 0,C 180,E1 -1251.842,E2 -1251.842} C_VEL
LIN {X 0,Y 594.342,Z 297.452,A -85,B 0,C 180,E1 -1253.891,E2 -1253.891} C_VEL
LIN {X 0,Y 594.333,Z 297.453,A -85,B 0,C 180,E1 -1255.931,E2 -1255.931} C_VEL
LIN {X 0,Y 594.371,Z 297.447,A -85,B 0,C 180,E1 -1257.967,E2 -1257.967} C_VEL
LIN {X 0,Y 594.389,Z 297.443,A -85,B 0,C 180,E1 -1260,E2 -1260} C_VEL
LIN {X 0,Y 594.362,Z 297.442,A -85,B 0,C 180,E1 -1262.711,E2 -1262.711} C_VEL
LIN {X 0,Y 594.373,Z 297.448,A -85,B 0,C 180,E1 -1265.428,E2 -1265.428} C_VEL
LIN {X 0,Y 594.36,Z 297.445,A -85,B 0,C 180,E1 -1268.158,E2 -1268.158} C_VEL
LIN {X 0,Y 594.357,Z 297.445,A -85,B 0,C 180,E1 -1271.062,E2 -1271.062} C_VEL
LIN {X 0,Y 594.355,Z 297.452,A -85,B 0,C 180,E1 -1273.68,E2 -1273.68} C_VEL
LIN {X 0,Y 594.325,Z 297.449,A -85,B 0,C 180,E1 -1275.284,E2 -1275.284} C_VEL
LIN {X 0,Y 593.653,Z 297.538,A -85,B 0,C 180,E1 -1275.85,E2 -1275.85} C_VEL
LIN {X 0,Y 590.787,Z 297.895,A -85,B 0,C 180,E1 -1276.768,E2 -1276.768} C_VEL
LIN {X 0,Y 588.374,Z 298.198,A -85,B 0,C 180,E1 -1277.506,E2 -1277.506} C_VEL
LIN {X 0,Y 587.349,Z 298.319,A -85,B 0,C 180,E1 -1278.076,E2 -1278.076} C_VEL
LIN {X 0,Y 587.272,Z 298.327,A -85,B 0,C 180,E1 -1278.269,E2 -1278.269} C_VEL
LIN {X 0,Y 587.323,Z 298.321,A -85,B 0,C 180,E1 -1281.038,E2 -1281.038} C_VEL
LIN {X 0,Y 587.278,Z 298.328,A -85,B 0,C 180,E1 -1284.009,E2 -1284.009} C_VEL
LIN {X 0,Y 587.292,Z 298.323,A -85,B 0,C 180,E1 -1286.281,E2 -1286.281} C_VEL
LIN {X 0,Y 587.332,Z 298.319,A -85,B 0,C 180,E1 -1289.132,E2 -1289.132} C_VEL
LIN {X 0,Y 587.307,Z 298.326,A -85,B 0,C 180,E1 -1291.831,E2 -1291.831} C_VEL
LIN {X 0,Y 587.319,Z 298.32,A -85,B 0,C 180,E1 -1294.345,E2 -1294.345} C_VEL
LIN {X 0,Y 587.325,Z 298.325,A -85,B 0,C 180,E1 -1297.609,E2 -1297.609} C_VEL
LIN {X 0,Y 587.286,Z 298.323,A -85,B 0,C 180,E1 -1300.257,E2 -1300.257} C_VEL
LIN {X 0,Y 587.29,Z 298.329,A -85,B 0,C 180,E1 -1303.117,E2 -1303.117} C_VEL
LIN {X 0,Y 587.291,Z 298.323,A -85,B 0,C 180,E1 -1306.047,E2 -1306.047} C_VEL
LIN {X 0,Y 587.3,Z 298.325,A -85,B 0,C 180,E1 -1308.929,E2 -1308.929} C_VEL
LIN {X 0,Y 587.304,Z 298.329,A -85,B 0,C 180,E1 -1311.519,E2 -1311.519} C_VEL
LIN {X 0,Y 587.274,Z 298.326,A -85,B 0,C 180,E1 -1314.099,E2 -1314.099} C_VEL
LIN {X 0,Y 587.307,Z 298.322,A -85,B 0,C 180,E1 -1316.602,E2 -1316.602} C_VEL
LIN {X 0,Y 587.302,Z 298.327,A -85,B 0,C 180,E1 -1319.032,E2 -1319.032} C_VEL
LIN {X 0,Y 587.296,Z 298.329,A -85,B 0,C 180,E1 -1321.402,E2 -1321.402} C_VEL
LIN {X 0,Y 587.293,Z 298.326,A -85,B 0,C 180,E1 -1323.833,E2 -1323.833} C_VEL
LIN {X 0,Y 587.294,Z 298.326,A -85,B 0,C 180,E1 -1326.741,E2 -1326.741} C_VEL
LIN {X 0,Y 587.309,Z 298.325,A -85,B 0,C 180,E1 -1329.695,E2 -1329.695} C_VEL
LIN {X 0,Y 587.278,Z 298.322,A -85,B 0,C 180,E1 -1331.872,E2 -1331.872} C_VEL
LIN {X 0,Y 587.289,Z 298.326,A -85,B 0,C 180,E1 -1334.024,E2 -1334.024} C_VEL
LIN {X 0,Y 587.372,Z 298.523,A -85,B 0,C 180,E1 -1336.772,E2 -1336.772} C_VEL
LIN {X 0,Y 587.655,Z 299.676,A -85,B 0,C 180,E1 -1336.88,E2 -1336.88} C_VEL
LIN {X 0,Y 587.832,Z 328.522,A -85,B 0,C 180,E1 -1337.244,E2 -1337.244} C_VEL
LIN {X 0,Y 587.742,Z 380.897,A -85,B 0,C 180,E1 -1337.899,E2 -1337.899} C_VEL
LIN {X 0,Y 587.704,Z 394.187,A -85,B 0,C 180,E1 -1338.205,E2 -1338.205} C_VEL
LIN {X 0,Y 587.629,Z 406.75,A -85,B 0,C 180,E1 -1338.635,E2 -1338.635} C_VEL
LIN {X 0,Y 587.57,Z 417.782,A -85,B 0,C 180,E1 -1339.142,E2 -1339.142} C_VEL
LIN {X 0,Y 587.477,Z 429.54,A -85,B 0,C 180,E1 -1339.837,E2 -1339.837} C_VEL
LIN {X 0,Y 587.393,Z 440.053,A -85,B 0,C 180,E1 -1340.618,E2 -1340.618} C_VEL
LIN {X 0,Y 587.323,Z 448.654,A -85,B 0,C 180,E1 -1341.398,E2 -1341.398} C_VEL
LIN {X 0,Y 587.274,Z 456.579,A -85,B 0,C 180,E1 -1342.263,E2 -1342.263} C_VEL
LIN {X 0,Y 587.235,Z 463.149,A -85,B 0,C 180,E1 -1343.127,E2 -1343.127} C_VEL
LIN {X 0,Y 587.237,Z 469.619,A -85,B 0,C 180,E1 -1344.161,E2 -1344.161} C_VEL
LIN {X 0,Y 587.147,Z 474.759,A -85,B 0,C 180,E1 -1345.194,E2 -1345.194} C_VEL
LIN {X 0,Y 587.213,Z 478.748,A -85,B 0,C 180,E1 -1346.226,E2 -1346.226} C_VEL
LIN {X 0,Y 587.131,Z 481.698,A -85,B 0,C 180,E1 -1347.256,E2 -1347.256} C_VEL
LIN {X 0,Y 587.14,Z 483.127,A -85,B 0,C 180,E1 -1347.942,E2 -1347.942} C_VEL
LIN {X 0,Y 587.14,Z 484.754,A -85,B 0,C 180,E1 -1349.314,E2 -1349.314} C_VEL
LIN {X 0,Y 587.137,Z 484.996,A -85,B 0,C 180,E1 -1350,E2 -1350} C_VEL
LIN {X 0,Y 587.14,Z 484.815,A -85,B 0,C 180,E1 -1350.686,E2 -1350.686} C_VEL
LIN {X 0,Y 587.141,Z 483.274,A -85,B 0,C 180,E1 -1352.058,E2 -1352.058} C_VEL
LIN {X 0,Y 587.133,Z 481.914,A -85,B 0,C 180,E1 -1352.744,E2 -1352.744} C_VEL
LIN {X 0,Y 587.213,Z 479.036,A -85,B 0,C 180,E1 -1353.774,E2 -1353.774} C_VEL
LIN {X 0,Y 587.147,Z 475.136,A -85,B 0,C 180,E1 -1354.806,E2 -1354.806} C_VEL
LIN {X 0,Y 587.229,Z 470.105,A -85,B 0,C 180,E1 -1355.839,E2 -1355.839} C_VEL
LIN {X 0,Y 587.23,Z 463.785,A -85,B 0,C 180,E1 -1356.874,E2 -1356.874} C_VEL
LIN {X 0,Y 587.288,Z 455.865,A -85,B 0,C 180,E1 -1357.91,E2 -1357.91} C_VEL
LIN {X 0,Y 587.343,Z 446.018,A -85,B 0,C 180,E1 -1358.949,E2 -1358.949} C_VEL
LIN {X 0,Y 587.421,Z 435.701,A -85,B 0,C 180,E1 -1359.816,E2 -1359.816} C_VEL
LIN {X 0,Y 587.531,Z 424.068,A -85,B 0,C 180,E1 -1360.598,E2 -1360.598} C_VEL
LIN {X 0,Y 587.575,Z 413.282,A -85,B 0,C 180,E1 -1361.172,E2 -1361.172} C_VEL
LIN {X 0,Y 587.632,Z 400.594,A -85,B 0,C 180,E1 -1361.685,E2 -1361.685} C_VEL
LIN {X 0,Y 587.716,Z 387.501,A -85,B 0,C 180,E1 -1362.057,E2 -1362.057} C_VEL
LIN {X 0,Y 587.785,Z 375.188,A -85,B 0,C 180,E1 -1362.275,E2 -1362.275} C_VEL
LIN {X 0,Y 587.762,Z 300.193,A -85,B 0,C 180,E1 -1363.197,E2 -1363.197} C_VEL
LIN {X 0,Y 587.408,Z 298.821,A -85,B 0,C 180,E1 -1363.271,E2 -1363.271} C_VEL
LIN {X 0,Y 587.302,Z 298.35,A -85,B 0,C 180,E1 -1363.406,E2 -1363.406} C_VEL
LIN {X 0,Y 587.283,Z 298.326,A -85,B 0,C 180,E1 -1365.976,E2 -1365.976} C_VEL
LIN {X 0,Y 587.315,Z 298.328,A -85,B 0,C 180,E1 -1369.031,E2 -1369.031} C_VEL
LIN {X 0,Y 587.295,Z 298.322,A -85,B 0,C 180,E1 -1371.775,E2 -1371.775} C_VEL
LIN {X 0,Y 587.282,Z 298.331,A -85,B 0,C 180,E1 -1374.564,E2 -1374.564} C_VEL
LIN {X 0,Y 587.293,Z 298.326,A -85,B 0,C 180,E1 -1377.048,E2 -1377.048} C_VEL
LIN {X 0,Y 587.299,Z 298.324,A -85,B 0,C 180,E1 -1379.382,E2 -1379.382} C_VEL
LIN {X 0,Y 587.313,Z 298.321,A -85,B 0,C 180,E1 -1381.83,E2 -1381.83} C_VEL
LIN {X 0,Y 587.326,Z 298.323,A -85,B 0,C 180,E1 -1384.344,E2 -1384.344} C_VEL
LIN {X 0,Y 587.3,Z 298.321,A -85,B 0,C 180,E1 -1387.61,E2 -1387.61} C_VEL
LIN {X 0,Y 587.291,Z 298.327,A -85,B 0,C 180,E1 -1390.255,E2 -1390.255} C_VEL
LIN {X 0,Y 587.282,Z 298.326,A -85,B 0,C 180,E1 -1393.114,E2 -1393.114} C_VEL
LIN {X 0,Y 587.281,Z 298.326,A -85,B 0,C 180,E1 -1396.045,E2 -1396.045} C_VEL
LIN {X 0,Y 587.303,Z 298.326,A -85,B 0,C 180,E1 -1398.928,E2 -1398.928} C_VEL
LIN {X 0,Y 587.293,Z 298.321,A -85,B 0,C 180,E1 -1401.518,E2 -1401.518} C_VEL
LIN {X 0,Y 587.265,Z 298.329,A -85,B 0,C 180,E1 -1404.098,E2 -1404.098} C_VEL
LIN {X 0,Y 587.324,Z 298.324,A -85,B 0,C 180,E1 -1406.889,E2 -1406.889} C_VEL
LIN {X 0,Y 587.28,Z 298.322,A -85,B 0,C 180,E1 -1409.498,E2 -1409.498} C_VEL
LIN {X 0,Y 587.277,Z 298.322,A -85,B 0,C 180,E1 -1411.4,E2 -1411.4} C_VEL
LIN {X 0,Y 587.304,Z 298.322,A -85,B 0,C 180,E1 -1413.828,E2 -1413.828} C_VEL
LIN {X 0,Y 587.28,Z 298.331,A -85,B 0,C 180,E1 -1416.739,E2 -1416.739} C_VEL
LIN {X 0,Y 587.293,Z 298.323,A -85,B 0,C 180,E1 -1419.694,E2 -1419.694} C_VEL
LIN {X 0,Y 587.268,Z 298.328,A -85,B 0,C 180,E1 -1421.871,E2 -1421.871} C_VEL
LIN {X 0,Y 587.293,Z 298.327,A -85,B 0,C 180,E1 -1424.736,E2 -1424.736} C_VEL
LIN {X 0,Y 587.267,Z 298.33,A -85,B 0,C 180,E1 -1426.857,E2 -1426.857} C_VEL
LIN {X 0,Y 587.328,Z 298.321,A -85,B 0,C 180,E1 -1428.962,E2 -1428.962} C_VEL
LIN {X 0,Y 587.306,Z 298.322,A -85,B 0,C 180,E1 -1431.744,E2 -1431.744} C_VEL
LIN {X 0,Y 587.334,Z 298.327,A -85,B 0,C 180,E1 -1434.507,E2 -1434.507} C_VEL
LIN {X 0,Y 587.332,Z 298.318,A -85,B 0,C 180,E1 -1437.257,E2 -1437.257} C_VEL
LIN {X 0,Y 587.355,Z 298.318,A -85,B 0,C 180,E1 -1440,E2 -1440} C_VEL
LIN {X 0,Y 587.354,Z 298.319,A -85,B 0,C 180,E1 -1442.743,E2 -1442.743} C_VEL
LIN {X 0,Y 587.313,Z 298.32,A -85,B 0,C 180,E1 -1445.493,E2 -1445.493} C_VEL
LIN {X 0,Y 587.293,Z 298.323,A -85,B 0,C 180,E1 -1447.564,E2 -1447.564} C_VEL
LIN {X 0,Y 587.317,Z 298.329,A -85,B 0,C 180,E1 -1450.34,E2 -1450.34} C_VEL
LIN {X 0,Y 587.285,Z 298.323,A -85,B 0,C 180,E1 -1453.142,E2 -1453.142} C_VEL
LIN {X 0,Y 587.304,Z 298.322,A -85,B 0,C 180,E1 -1455.264,E2 -1455.264} C_VEL
LIN {X 0,Y 587.272,Z 298.326,A -85,B 0,C 180,E1 -1457.408,E2 -1457.408} C_VEL
LIN {X 0,Y 587.293,Z 298.323,A -85,B 0,C 180,E1 -1459.577,E2 -1459.577} C_VEL
LIN {X 0,Y 587.302,Z 298.323,A -85,B 0,C 180,E1 -1461.775,E2 -1461.775} C_VEL
LIN {X 0,Y 587.299,Z 298.324,A -85,B 0,C 180,E1 -1464.761,E2 -1464.761} C_VEL
LIN {X 0,Y 587.293,Z 298.325,A -85,B 0,C 180,E1 -1467.684,E2 -1467.684} C_VEL
LIN {X 0,Y 587.321,Z 298.33,A -85,B 0,C 180,E1 -1470.171,E2 -1470.171} C_VEL
LIN {X 0,Y 587.327,Z 298.319,A -85,B 0,C 180,E1 -1473.111,E2 -1473.111} C_VEL
LIN {X 0,Y 587.269,Z 298.332,A -85,B 0,C 180,E1 -1475.902,E2 -1475.902} C_VEL
LIN {X 0,Y 587.307,Z 298.325,A -85,B 0,C 180,E1 -1478.481,E2 -1478.481} C_VEL
LIN {X 0,Y 587.299,Z 298.323,A -85,B 0,C 180,E1 -1481.16,E2 -1481.16} C_VEL
LIN {X 0,Y 587.294,Z 298.331,A -85,B 0,C 180,E1 -1483.953,E2 -1483.953} C_VEL
LIN {X 0,Y 587.277,Z 298.325,A -85,B 0,C 180,E1 -1486.886,E2 -1486.886} C_VEL
LIN {X 0,Y 587.298,Z 298.328,A -85,B 0,C 180,E1 -1489.745,E2 -1489.745} C_VEL
LIN {X 0,Y 587.313,Z 298.325,A -85,B 0,C 180,E1 -1492.391,E2 -1492.391} C_VEL
LIN {X 0,Y 587.324,Z 298.324,A -85,B 0,C 180,E1 -1495.656,E2 -1495.656} C_VEL
LIN {X 0,Y 587.33,Z 298.325,A -85,B 0,C 180,E1 -1498.231,E2 -1498.231} C_VEL
LIN {X 0,Y 587.298,Z 298.322,A -85,B 0,C 180,E1 -1500.876,E2 -1500.876} C_VEL
LIN {X 0,Y 587.336,Z 298.516,A -85,B 0,C 180,E1 -1503.195,E2 -1503.195} C_VEL
LIN {X 0,Y 588.416,Z 303.361,A -85,B 0,C 180,E1 -1503.774,E2 -1503.774} C_VEL
LIN {X 0,Y 588.241,Z 325.349,A -85,B 0,C 180,E1 -1506.22,E2 -1506.22} C_VEL
LIN {X 0,Y 587.982,Z 352.244,A -85,B 0,C 180,E1 -1509.171,E2 -1509.171} C_VEL
LIN {X 0,Y 587.774,Z 379.14,A -85,B 0,C 180,E1 -1512.068,E2 -1512.068} C_VEL
LIN {X 0,Y 587.615,Z 404.355,A -85,B 0,C 180,E1 -1514.745,E2 -1514.745} C_VEL
LIN {X 0,Y 587.496,Z 420.896,A -85,B 0,C 180,E1 -1516.466,E2 -1516.466} C_VEL
LIN {X 0,Y 587.897,Z 424.95,A -85,B 0,C 180,E1 -1516.542,E2 -1516.542} C_VEL
LIN {X 0,Y 587.746,Z 530.958,A -85,B 0,C 180,E1 -1517.856,E2 -1517.856} C_VEL
LIN {X 0,Y 587.694,Z 543.465,A -85,B 0,C 180,E1 -1518.139,E2 -1518.139} C_VEL
LIN {X 0,Y 587.612,Z 555.58,A -85,B 0,C 180,E1 -1518.544,E2 -1518.544} C_VEL
LIN {X 0,Y 587.543,Z 566.931,A -85,B 0,C 180,E1 -1519.054,E2 -1519.054} C_VEL
LIN {X 0,Y 587.465,Z 577.586,A -85,B 0,C 180,E1 -1519.663,E2 -1519.663} C_VEL
LIN {X 0,Y 587.391,Z 588.477,A -85,B 0,C 180,E1 -1520.444,E2 -1520.444} C_VEL
LIN {X 0,Y 587.321,Z 599.114,A -85,B 0,C 180,E1 -1521.398,E2 -1521.398} C_VEL
LIN {X 0,Y 587.273,Z 606.962,A -85,B 0,C 180,E1 -1522.263,E2 -1522.263} C_VEL
LIN {X 0,Y 587.23,Z 613.47,A -85,B 0,C 180,E1 -1523.126,E2 -1523.126} C_VEL
LIN {X 0,Y 587.236,Z 619.867,A -85,B 0,C 180,E1 -1524.161,E2 -1524.161} C_VEL
LIN {X 0,Y 587.147,Z 624.95,A -85,B 0,C 180,E1 -1525.194,E2 -1525.194} C_VEL
LIN {X 0,Y 587.212,Z 628.896,A -85,B 0,C 180,E1 -1526.226,E2 -1526.226} C_VEL
LIN {X 0,Y 587.132,Z 631.809,A -85,B 0,C 180,E1 -1527.256,E2 -1527.256} C_VEL
LIN {X 0,Y 587.139,Z 633.2,A -85,B 0,C 180,E1 -1527.942,E2 -1527.942} C_VEL
LIN {X 0,Y 587.14,Z 634.784,A -85,B 0,C 180,E1 -1529.314,E2 -1529.314} C_VEL
LIN {X 0,Y 587.137,Z 635,A -85,B 0,C 180,E1 -1530,E2 -1530} C_VEL
LIN {X 0,Y 587.147,Z 634.185,A -85,B 0,C 180,E1 -1531.372,E2 -1531.372} C_VEL
LIN {X 0,Y 587.139,Z 633.201,A -85,B 0,C 180,E1 -1532.058,E2 -1532.058} C_VEL
LIN {X 0,Y 587.132,Z 631.81,A -85,B 0,C 180,E1 -1532.744,E2 -1532.744} C_VEL
LIN {X 0,Y 587.212,Z 628.896,A -85,B 0,C 180,E1 -1533.774,E2 -1533.774} C_VEL
LIN {X 0,Y 587.147,Z 624.95,A -85,B 0,C 180,E1 -1534.806,E2 -1534.806} C_VEL
LIN {X 0,Y 587.217,Z 618.878,A -85,B 0,C 180,E1 -1536.011,E2 -1536.011} C_VEL
LIN {X 0,Y 587.245,Z 612.238,A -85,B 0,C 180,E1 -1537.046,E2 -1537.046} C_VEL
LIN {X 0,Y 587.299,Z 603.991,A -85,B 0,C 180,E1 -1538.083,E2 -1538.083} C_VEL
LIN {X 0,Y 587.343,Z 595.539,A -85,B 0,C 180,E1 -1538.949,E2 -1538.949} C_VEL
LIN {X 0,Y 587.416,Z 585.098,A -85,B 0,C 180,E1 -1539.816,E2 -1539.816} C_VEL
LIN {X 0,Y 587.49,Z 574.761,A -85,B 0,C 180,E1 -1540.511,E2 -1540.511} C_VEL
LIN {X 0,Y 587.584,Z 562.804,A -85,B 0,C 180,E1 -1541.149,E2 -1541.149} C_VEL
LIN {X 0,Y 587.631,Z 550.596,A -85,B 0,C 180,E1 -1541.639,E2 -1541.639} C_VEL
LIN {X 0,Y 587.707,Z 537.445,A -85,B 0,C 180,E1 -1542.014,E2 -1542.014} C_VEL
LIN {X 0,Y 587.747,Z 525.101,A -85,B 0,C 180,E1 -1542.232,E2 -1542.232} C_VEL
LIN {X 0,Y 587.811,Z 423.163,A -85,B 0,C 180,E1 -1543.482,E2 -1543.482} C_VEL
LIN {X 0,Y 587.492,Z 420.576,A -85,B 0,C 180,E1 -1543.556,E2 -1543.556} C_VEL
LIN {X 0,Y 587.681,Z 394.269,A -85,B 0,C 180,E1 -1546.322,E2 -1546.322} C_VEL
LIN {X 0,Y 587.864,Z 366.348,A -85,B 0,C 180,E1 -1549.304,E2 -1549.304} C_VEL
LIN {X 0,Y 588.08,Z 340.478,A -85,B 0,C 180,E1 -1552.113,E2 -1552.113} C_VEL
LIN {X 0,Y 588.35,Z 315.433,A -85,B 0,C 180,E1 -1554.883,E2 -1554.883} C_VEL
LIN {X 0,Y 588.46,Z 303.366,A -85,B 0,C 180,E1 -1556.224,E2 -1556.224} C_VEL
LIN {X 0,Y 587.322,Z 298.425,A -85,B 0,C 180,E1 -1556.83,E2 -1556.83} C_VEL
LIN {X 0,Y 587.299,Z 298.323,A -85,B 0,C 180,E1 -1559.382,E2 -1559.382} C_VEL
LIN {X 0,Y 587.312,Z 298.328,A -85,B 0,C 180,E1 -1561.83,E2 -1561.83} C_VEL
LIN {X 0,Y 587.324,Z 298.325,A -85,B 0,C 180,E1 -1564.344,E2 -1564.344} C_VEL
LIN {X 0,Y 587.314,Z 298.325,A -85,B 0,C 180,E1 -1567.609,E2 -1567.609} C_VEL
LIN {X 0,Y 587.298,Z 298.329,A -85,B 0,C 180,E1 -1570.255,E2 -1570.255} C_VEL
LIN {X 0,Y 587.277,Z 298.325,A -85,B 0,C 180,E1 -1573.114,E2 -1573.114} C_VEL
LIN {X 0,Y 587.294,Z 298.332,A -85,B 0,C 180,E1 -1576.047,E2 -1576.047} C_VEL
LIN {X 0,Y 587.3,Z 298.323,A -85,B 0,C 180,E1 -1578.84,E2 -1578.84} C_VEL
LIN {X 0,Y 587.307,Z 298.324,A -85,B 0,C 180,E1 -1581.519,E2 -1581.519} C_VEL
LIN {X 0,Y 587.269,Z 298.331,A -85,B 0,C 180,E1 -1584.098,E2 -1584.098} C_VEL
LIN {X 0,Y 587.327,Z 298.319,A -85,B 0,C 180,E1 -1586.889,E2 -1586.889} C_VEL
LIN {X 0,Y 587.334,Z 298.328,A -85,B 0,C 180,E1 -1589.83,E2 -1589.83} C_VEL
LIN {X 0,Y 587.292,Z 298.326,A -85,B 0,C 180,E1 -1592.316,E2 -1592.316} C_VEL
LIN {X 0,Y 587.299,Z 298.324,A -85,B 0,C 180,E1 -1595.239,E2 -1595.239} C_VEL
LIN {X 0,Y 587.303,Z 298.324,A -85,B 0,C 180,E1 -1598.225,E2 -1598.225} C_VEL
LIN {X 0,Y 587.33,Z 298.319,A -85,B 0,C 180,E1 -1601.151,E2 -1601.151} C_VEL
LIN {X 0,Y 587.296,Z 298.329,A -85,B 0,C 180,E1 -1604.024,E2 -1604.024} C_VEL
LIN {X 0,Y 587.329,Z 298.322,A -85,B 0,C 180,E1 -1606.154,E2 -1606.154} C_VEL
LIN {X 0,Y 587.328,Z 298.319,A -85,B 0,C 180,E1 -1608.962,E2 -1608.962} C_VEL
LIN {X 0,Y 587.313,Z 298.331,A -85,B 0,C 180,E1 -1611.744,E2 -1611.744} C_VEL
LIN {X 0,Y 587.3,Z 298.331,A -85,B 0,C 180,E1 -1613.817,E2 -1613.817} C_VEL
LIN {X 0,Y 587.289,Z 298.331,A -85,B 0,C 180,E1 -1615.883,E2 -1615.883} C_VEL
LIN {X 0,Y 587.343,Z 298.323,A -85,B 0,C 180,E1 -1617.943,E2 -1617.943} C_VEL
LIN {X 0,Y 587.359,Z 298.319,A -85,B 0,C 180,E1 -1620,E2 -1620} C_VEL
LIN {X 0,Y 587.332,Z 298.318,A -85,B 0,C 180,E1 -1622.743,E2 -1622.743} C_VEL
LIN {X 0,Y 587.337,Z 298.325,A -85,B 0,C 180,E1 -1625.493,E2 -1625.493} C_VEL
LIN {X 0,Y 587.32,Z 298.32,A -85,B 0,C 180,E1 -1628.256,E2 -1628.256} C_VEL
LIN {X 0,Y 587.321,Z 298.322,A -85,B 0,C 180,E1 -1631.125,E2 -1631.125} C_VEL
LIN {X 0,Y 587.308,Z 298.321,A -85,B 0,C 180,E1 -1634.242,E2 -1634.242} C_VEL
LIN {X 0,Y 587.299,Z 298.323,A -85,B 0,C 180,E1 -1636.801,E2 -1636.801} C_VEL
LIN {X 0,Y 587.272,Z 298.327,A -85,B 0,C 180,E1 -1638.269,E2 -1638.269} C_VEL
LIN {X 0,Y 586.635,Z 298.406,A -85,B 0,C 180,E1 -1638.841,E2 -1638.841} C_VEL
LIN {X 0,Y 583.835,Z 298.76,A -85,B 0,C 180,E1 -1639.77,E2 -1639.77} C_VEL
LIN {X 0,Y 581.438,Z 299.054,A -85,B 0,C 180,E1 -1640.517,E2 -1640.517} C_VEL
LIN {X 0,Y 580.378,Z 299.187,A -85,B 0,C 180,E1 -1641.094,E2 -1641.094} C_VEL
LIN {X 0,Y 580.276,Z 299.202,A -85,B 0,C 180,E1 -1641.289,E2 -1641.289} C_VEL
LIN {X 0,Y 580.241,Z 299.212,A -85,B 0,C 180,E1 -1643.56,E2 -1643.56} C_VEL
LIN {X 0,Y 580.253,Z 299.199,A -85,B 0,C 180,E1 -1646.328,E2 -1646.328} C_VEL
LIN {X 0,Y 580.265,Z 299.202,A -85,B 0,C 180,E1 -1649.305,E2 -1649.305} C_VEL
LIN {X 0,Y 580.275,Z 299.197,A -85,B 0,C 180,E1 -1652.202,E2 -1652.202} C_VEL
LIN {X 0,Y 580.267,Z 299.199,A -85,B 0,C 180,E1 -1654.698,E2 -1654.698} C_VEL
LIN {X 0,Y 580.275,Z 299.204,A -85,B 0,C 180,E1 -1657.27,E2 -1657.27} C_VEL
LIN {X 0,Y 580.267,Z 299.197,A -85,B 0,C 180,E1 -1660.269,E2 -1660.269} C_VEL
LIN {X 0,Y 580.233,Z 299.213,A -85,B 0,C 180,E1 -1663.387,E2 -1663.387} C_VEL
LIN {X 0,Y 580.23,Z 299.201,A -85,B 0,C 180,E1 -1666.339,E2 -1666.339} C_VEL
LIN {X 0,Y 580.27,Z 299.204,A -85,B 0,C 180,E1 -1669.155,E2 -1669.155} C_VEL
LIN {X 0,Y 580.27,Z 299.199,A -85,B 0,C 180,E1 -1671.93,E2 -1671.93} C_VEL
LIN {X 0,Y 580.227,Z 299.204,A -85,B 0,C 180,E1 -1674.452,E2 -1674.452} C_VEL
LIN {X 0,Y 580.259,Z 299.204,A -85,B 0,C 180,E1 -1676.974,E2 -1676.974} C_VEL
LIN {X 0,Y 580.265,Z 299.208,A -85,B 0,C 180,E1 -1679.424,E2 -1679.424} C_VEL
LIN {X 0,Y 580.244,Z 299.198,A -85,B 0,C 180,E1 -1682.152,E2 -1682.152} C_VEL
LIN {X 0,Y 580.235,Z 299.207,A -85,B 0,C 180,E1 -1684.917,E2 -1684.917} C_VEL
LIN {X 0,Y 580.277,Z 299.206,A -85,B 0,C 180,E1 -1687.197,E2 -1687.197} C_VEL
LIN {X 0,Y 580.263,Z 299.207,A -85,B 0,C 180,E1 -1689.437,E2 -1689.437} C_VEL
LIN {X 0,Y 580.242,Z 299.199,A -85,B 0,C 180,E1 -1691.645,E2 -1691.645} C_VEL
LIN {X 0,Y 580.246,Z 299.205,A -85,B 0,C 180,E1 -1693.825,E2 -1693.825} C_VEL
LIN {X 0,Y 580.305,Z 299.36,A -85,B 0,C 180,E1 -1696.608,E2 -1696.608} C_VEL
LIN {X 0,Y 580.496,Z 300.242,A -85,B 0,C 180,E1 -1696.712,E2 -1696.712} C_VEL
LIN {X 0,Y 580.937,Z 301.742,A -85,B 0,C 180,E1 -1696.756,E2 -1696.756} C_VEL
LIN {X 0,Y 580.824,Z 380.926,A -85,B 0,C 180,E1 -1697.753,E2 -1697.753} C_VEL
LIN {X 0,Y 580.757,Z 394.206,A -85,B 0,C 180,E1 -1698.062,E2 -1698.062} C_VEL
LIN {X 0,Y 580.677,Z 406.366,A -85,B 0,C 180,E1 -1698.481,E2 -1698.481} C_VEL
LIN {X 0,Y 580.593,Z 417.795,A -85,B 0,C 180,E1 -1699.009,E2 -1699.009} C_VEL
LIN {X 0,Y 580.457,Z 429.546,A -85,B 0,C 180,E1 -1699.713,E2 -1699.713} C_VEL
LIN {X 0,Y 580.345,Z 440.061,A -85,B 0,C 180,E1 -1700.503,E2 -1700.503} C_VEL
LIN {X 0,Y 580.272,Z 448.661,A -85,B 0,C 180,E1 -1701.292,E2 -1701.292} C_VEL
LIN {X 0,Y 580.222,Z 456.583,A -85,B 0,C 180,E1 -1702.168,E2 -1702.168} C_VEL
LIN {X 0,Y 580.168,Z 464.285,A -85,B 0,C 180,E1 -1703.21,E2 -1703.21} C_VEL
LIN {X 0,Y 580.165,Z 469.622,A -85,B 0,C 180,E1 -1704.09,E2 -1704.09} C_VEL
LIN {X 0,Y 580.054,Z 474.761,A -85,B 0,C 180,E1 -1705.135,E2 -1705.135} C_VEL
LIN {X 0,Y 580.109,Z 478.75,A -85,B 0,C 180,E1 -1706.18,E2 -1706.18} C_VEL
LIN {X 0,Y 580.043,Z 481.7,A -85,B 0,C 180,E1 -1707.222,E2 -1707.222} C_VEL
LIN {X 0,Y 580.04,Z 483.127,A -85,B 0,C 180,E1 -1707.917,E2 -1707.917} C_VEL
LIN {X 0,Y 580.041,Z 484.755,A -85,B 0,C 180,E1 -1709.306,E2 -1709.306} C_VEL
LIN {X 0,Y 580.038,Z 484.996,A -85,B 0,C 180,E1 -1710,E2 -1710} C_VEL
LIN {X 0,Y 580.04,Z 484.815,A -85,B 0,C 180,E1 -1710.694,E2 -1710.694} C_VEL
LIN {X 0,Y 580.04,Z 483.273,A -85,B 0,C 180,E1 -1712.083,E2 -1712.083} C_VEL
LIN {X 0,Y 580.044,Z 481.912,A -85,B 0,C 180,E1 -1712.778,E2 -1712.778} C_VEL
LIN {X 0,Y 580.11,Z 479.033,A -85,B 0,C 180,E1 -1713.821,E2 -1713.821} C_VEL
LIN {X 0,Y 580.054,Z 475.134,A -85,B 0,C 180,E1 -1714.865,E2 -1714.865} C_VEL
LIN {X 0,Y 580.162,Z 470.103,A -85,B 0,C 180,E1 -1715.91,E2 -1715.91} C_VEL
LIN {X 0,Y 580.158,Z 463.781,A -85,B 0,C 180,E1 -1716.958,E2 -1716.958} C_VEL
LIN {X 0,Y 580.241,Z 455.86,A -85,B 0,C 180,E1 -1718.007,E2 -1718.007} C_VEL
LIN {X 0,Y 580.308,Z 446.011,A -85,B 0,C 180,E1 -1719.058,E2 -1719.058} C_VEL
LIN {X 0,Y 580.421,Z 435.696,A -85,B 0,C 180,E1 -1719.936,E2 -1719.936} C_VEL
LIN {X 0,Y 580.543,Z 424.056,A -85,B 0,C 180,E1 -1720.727,E2 -1720.727} C_VEL
LIN {X 0,Y 580.612,Z 412.506,A -85,B 0,C 180,E1 -1721.343,E2 -1721.343} C_VEL
LIN {X 0,Y 580.705,Z 400.508,A -85,B 0,C 180,E1 -1721.828,E2 -1721.828} C_VEL
LIN {X 0,Y 580.785,Z 387.477,A -85,B 0,C 180,E1 -1722.203,E2 -1722.203} C_VEL
LIN {X 0,Y 580.855,Z 375.148,A -85,B 0,C 180,E1 -1722.424,E2 -1722.424} C_VEL
LIN {X 0,Y 580.798,Z 301.299,A -85,B 0,C 180,E1 -1723.343,E2 -1723.343} C_VEL
LIN {X 0,Y 580.379,Z 299.801,A -85,B 0,C 180,E1 -1723.413,E2 -1723.413} C_VEL
LIN {X 0,Y 580.271,Z 299.221,A -85,B 0,C 180,E1 -1723.571,E2 -1723.571} C_VEL
LIN {X 0,Y 580.239,Z 299.205,A -85,B 0,C 180,E1 -1726.175,E2 -1726.175} C_VEL
LIN {X 0,Y 580.267,Z 299.204,A -85,B 0,C 180,E1 -1729.141,E2 -1729.141} C_VEL
LIN {X 0,Y 580.281,Z 299.199,A -85,B 0,C 180,E1 -1731.305,E2 -1731.305} C_VEL
LIN {X 0,Y 580.24,Z 299.202,A -85,B 0,C 180,E1 -1733.559,E2 -1733.559} C_VEL
LIN {X 0,Y 580.247,Z 299.204,A -85,B 0,C 180,E1 -1736.324,E2 -1736.324} C_VEL
LIN {X 0,Y 580.259,Z 299.202,A -85,B 0,C 180,E1 -1739.302,E2 -1739.302} C_VEL
LIN {X 0,Y 580.276,Z 299.199,A -85,B 0,C 180,E1 -1742.201,E2 -1742.201} C_VEL
LIN {X 0,Y 580.275,Z 299.208,A -85,B 0,C 180,E1 -1744.697,E2 -1744.697} C_VEL
LIN {X 0,Y 580.262,Z 299.199,A -85,B 0,C 180,E1 -1747.27,E2 -1747.27} C_VEL
LIN {X 0,Y 580.272,Z 299.202,A -85,B 0,C 180,E1 -1750.268,E2 -1750.268} C_VEL
LIN {X 0,Y 580.226,Z 299.202,A -85,B 0,C 180,E1 -1753.385,E2 -1753.385} C_VEL
LIN {X 0,Y 580.222,Z 299.209,A -85,B 0,C 180,E1 -1756.336,E2 -1756.336} C_VEL
LIN {X 0,Y 580.25,Z 299.201,A -85,B 0,C 180,E1 -1759.152,E2 -1759.152} C_VEL
LIN {X 0,Y 580.269,Z 299.196,A -85,B 0,C 180,E1 -1761.928,E2 -1761.928} C_VEL
LIN {X 0,Y 580.217,Z 299.212,A -85,B 0,C 180,E1 -1764.45,E2 -1764.45} C_VEL
LIN {X 0,Y 580.274,Z 299.2,A -85,B 0,C 180,E1 -1766.974,E2 -1766.974} C_VEL
LIN {X 0,Y 580.246,Z 299.197,A -85,B 0,C 180,E1 -1769.422,E2 -1769.422} C_VEL
LIN {X 0,Y 580.232,Z 299.203,A -85,B 0,C 180,E1 -1772.152,E2 -1772.152} C_VEL
LIN {X 0,Y 580.27,Z 299.202,A -85,B 0,C 180,E1 -1774.918,E2 -1774.918} C_VEL
LIN {X 0,Y 580.225,Z 299.205,A -85,B 0,C 180,E1 -1777.945,E2 -1777.945} C_VEL
LIN {X 0,Y 580.27,Z 299.202,A -85,B 0,C 180,E1 -1780.912,E2 -1780.912} C_VEL
LIN {X 0,Y 580.228,Z 299.204,A -85,B 0,C 180,E1 -1783.824,E2 -1783.824} C_VEL
LIN {X 0,Y 580.271,Z 299.199,A -85,B 0,C 180,E1 -1785.982,E2 -1785.982} C_VEL
LIN {X 0,Y 580.297,Z 299.199,A -85,B 0,C 180,E1 -1788.827,E2 -1788.827} C_VEL
LIN {X 0,Y 580.278,Z 299.196,A -85,B 0,C 180,E1 -1791.643,E2 -1791.643} C_VEL
LIN {X 0,Y 580.298,Z 299.204,A -85,B 0,C 180,E1 -1794.44,E2 -1794.44} C_VEL
LIN {X 0,Y 580.302,Z 299.194,A -85,B 0,C 180,E1 -1797.223,E2 -1797.223} C_VEL
LIN {X 0,Y 580.325,Z 299.194,A -85,B 0,C 180,E1 -1800,E2 -1800} C_VEL
LIN {X 0,Y 580.318,Z 299.195,A -85,B 0,C 180,E1 -1802.777,E2 -1802.777} C_VEL
LIN {X 0,Y 580.283,Z 299.196,A -85,B 0,C 180,E1 -1805.56,E2 -1805.56} C_VEL
LIN {X 0,Y 580.245,Z 299.202,A -85,B 0,C 180,E1 -1807.656,E2 -1807.656} C_VEL
LIN {X 0,Y 580.27,Z 299.205,A -85,B 0,C 180,E1 -1810.467,E2 -1810.467} C_VEL
LIN {X 0,Y 580.281,Z 299.2,A -85,B 0,C 180,E1 -1812.592,E2 -1812.592} C_VEL
LIN {X 0,Y 580.271,Z 299.201,A -85,B 0,C 180,E1 -1814.735,E2 -1814.735} C_VEL
LIN {X 0,Y 580.237,Z 299.204,A -85,B 0,C 180,E1 -1817.626,E2 -1817.626} C_VEL
LIN {X 0,Y 580.27,Z 299.2,A -85,B 0,C 180,E1 -1819.824,E2 -1819.824} C_VEL
LIN {X 0,Y 580.254,Z 299.205,A -85,B 0,C 180,E1 -1822.053,E2 -1822.053} C_VEL
LIN {X 0,Y 580.267,Z 299.199,A -85,B 0,C 180,E1 -1825.082,E2 -1825.082} C_VEL
LIN {X 0,Y 580.269,Z 299.206,A -85,B 0,C 180,E1 -1828.187,E2 -1828.187} C_VEL
LIN {X 0,Y 580.271,Z 299.2,A -85,B 0,C 180,E1 -1830.694,E2 -1830.694} C_VEL
LIN {X 0,Y 580.274,Z 299.198,A -85,B 0,C 180,E1 -1833.313,E2 -1833.313} C_VEL
LIN {X 0,Y 580.217,Z 299.208,A -85,B 0,C 180,E1 -1835.754,E2 -1835.754} C_VEL
LIN {X 0,Y 580.272,Z 299.207,A -85,B 0,C 180,E1 -1838.148,E2 -1838.148} C_VEL
LIN {X 0,Y 580.269,Z 299.199,A -85,B 0,C 180,E1 -1840.846,E2 -1840.846} C_VEL
LIN {X 0,Y 580.229,Z 299.204,A -85,B 0,C 180,E1 -1843.387,E2 -1843.387} C_VEL
LIN {X 0,Y 580.23,Z 299.208,A -85,B 0,C 180,E1 -1846.339,E2 -1846.339} C_VEL
LIN {X 0,Y 580.271,Z 299.198,A -85,B 0,C 180,E1 -1849.155,E2 -1849.155} C_VEL
LIN {X 0,Y 580.275,Z 299.206,A -85,B 0,C 180,E1 -1851.929,E2 -1851.929} C_VEL
LIN {X 0,Y 580.221,Z 299.207,A -85,B 0,C 180,E1 -1854.451,E2 -1854.451} C_VEL
LIN {X 0,Y 580.24,Z 299.201,A -85,B 0,C 180,E1 -1856.973,E2 -1856.973} C_VEL
LIN {X 0,Y 580.277,Z 299.2,A -85,B 0,C 180,E1 -1859.425,E2 -1859.425} C_VEL
LIN {X 0,Y 580.247,Z 299.209,A -85,B 0,C 180,E1 -1862.151,E2 -1862.151} C_VEL
LIN {X 0,Y 580.287,Z 299.42,A -85,B 0,C 180,E1 -1863.038,E2 -1863.038} C_VEL
LIN {X 0,Y 581.46,Z 304.393,A -85,B 0,C 180,E1 -1863.639,E2 -1863.639} C_VEL
LIN {X 0,Y 581.458,Z 325.349,A -85,B 0,C 180,E1 -1865.926,E2 -1865.926} C_VEL
LIN {X 0,Y 581.153,Z 352.244,A -85,B 0,C 180,E1 -1868.914,E2 -1868.914} C_VEL
LIN {X 0,Y 580.853,Z 379.14,A -85,B 0,C 180,E1 -1871.847,E2 -1871.847} C_VEL
LIN {X 0,Y 580.634,Z 404.355,A -85,B 0,C 180,E1 -1874.557,E2 -1874.557} C_VEL
LIN {X 0,Y 580.515,Z 420.894,A -85,B 0,C 180,E1 -1876.301,E2 -1876.301} C_VEL
LIN {X 0,Y 580.997,Z 424.95,A -85,B 0,C 180,E1 -1876.379,E2 -1876.379} C_VEL
LIN {X 0,Y 580.81,Z 530.957,A -85,B 0,C 180,E1 -1877.708,E2 -1877.708} C_VEL
LIN {X 0,Y 580.756,Z 544.227,A -85,B 0,C 180,E1 -1878.018,E2 -1878.018} C_VEL
LIN {X 0,Y 580.658,Z 556.378,A -85,B 0,C 180,E1 -1878.436,E2 -1878.436} C_VEL
LIN {X 0,Y 580.564,Z 568.633,A -85,B 0,C 180,E1 -1879.009,E2 -1879.009} C_VEL
LIN {X 0,Y 580.423,Z 580.206,A -85,B 0,C 180,E1 -1879.712,E2 -1879.712} C_VEL
LIN {X 0,Y 580.341,Z 590.601,A -85,B 0,C 180,E1 -1880.503,E2 -1880.503} C_VEL
LIN {X 0,Y 580.271,Z 599.114,A -85,B 0,C 180,E1 -1881.292,E2 -1881.292} C_VEL
LIN {X 0,Y 580.221,Z 606.962,A -85,B 0,C 180,E1 -1882.168,E2 -1882.168} C_VEL
LIN {X 0,Y 580.153,Z 614.651,A -85,B 0,C 180,E1 -1883.222,E2 -1883.222} C_VEL
LIN {X 0,Y 580.139,Z 621.681,A -85,B 0,C 180,E1 -1884.439,E2 -1884.439} C_VEL
LIN {X 0,Y 580.108,Z 626.372,A -85,B 0,C 180,E1 -1885.484,E2 -1885.484} C_VEL
LIN {X 0,Y 580.123,Z 629.957,A -85,B 0,C 180,E1 -1886.527,E2 -1886.527} C_VEL
LIN {X 0,Y 580.043,Z 631.808,A -85,B 0,C 180,E1 -1887.222,E2 -1887.222} C_VEL
LIN {X 0,Y 580.038,Z 633.199,A -85,B 0,C 180,E1 -1887.917,E2 -1887.917} C_VEL
LIN {X 0,Y 580.04,Z 634.785,A -85,B 0,C 180,E1 -1889.306,E2 -1889.306} C_VEL
LIN {X 0,Y 580.037,Z 635,A -85,B 0,C 180,E1 -1890,E2 -1890} C_VEL
LIN {X 0,Y 580.047,Z 634.186,A -85,B 0,C 180,E1 -1891.389,E2 -1891.389} C_VEL
LIN {X 0,Y 580.038,Z 633.2,A -85,B 0,C 180,E1 -1892.083,E2 -1892.083} C_VEL
LIN {X 0,Y 580.043,Z 631.81,A -85,B 0,C 180,E1 -1892.778,E2 -1892.778} C_VEL
LIN {X 0,Y 580.109,Z 628.896,A -85,B 0,C 180,E1 -1893.82,E2 -1893.82} C_VEL
LIN {X 0,Y 580.054,Z 624.95,A -85,B 0,C 180,E1 -1894.865,E2 -1894.865} C_VEL
LIN {X 0,Y 580.139,Z 618.878,A -85,B 0,C 180,E1 -1896.085,E2 -1896.085} C_VEL
LIN {X 0,Y 580.184,Z 612.238,A -85,B 0,C 180,E1 -1897.132,E2 -1897.132} C_VEL
LIN {X 0,Y 580.25,Z 603.992,A -85,B 0,C 180,E1 -1898.182,E2 -1898.182} C_VEL
LIN {X 0,Y 580.308,Z 595.54,A -85,B 0,C 180,E1 -1899.058,E2 -1899.058} C_VEL
LIN {X 0,Y 580.417,Z 585.099,A -85,B 0,C 180,E1 -1899.936,E2 -1899.936} C_VEL
LIN {X 0,Y 580.495,Z 574.759,A -85,B 0,C 180,E1 -1900.639,E2 -1900.639} C_VEL
LIN {X 0,Y 580.597,Z 563.235,A -85,B 0,C 180,E1 -1901.264,E2 -1901.264} C_VEL
LIN {X 0,Y 580.669,Z 550.478,A -85,B 0,C 180,E1 -1901.785,E2 -1901.785} C_VEL
LIN {X 0,Y 580.754,Z 537.444,A -85,B 0,C 180,E1 -1902.16,E2 -1902.16} C_VEL
LIN {X 0,Y 580.837,Z 525.101,A -85,B 0,C 180,E1 -1902.38,E2 -1902.38} C_VEL
LIN {X 0,Y 580.794,Z 423.163,A -85,B 0,C 180,E1 -1903.648,E2 -1903.648} C_VEL
LIN {X 0,Y 580.515,Z 420.579,A -85,B 0,C 180,E1 -1903.722,E2 -1903.722} C_VEL
LIN {X 0,Y 580.734,Z 394.269,A -85,B 0,C 180,E1 -1906.522,E2 -1906.522} C_VEL
LIN {X 0,Y 580.951,Z 366.746,A -85,B 0,C 180,E1 -1909.5,E2 -1909.5} C_VEL
LIN {X 0,Y 581.231,Z 342.159,A -85,B 0,C 180,E1 -1912.201,E2 -1912.201} C_VEL
LIN {X 0,Y 581.511,Z 318.252,A -85,B 0,C 180,E1 -1914.857,E2 -1914.857} C_VEL
LIN {X 0,Y 581.493,Z 304.388,A -85,B 0,C 180,E1 -1916.361,E2 -1916.361} C_VEL
LIN {X 0,Y 580.275,Z 299.329,A -85,B 0,C 180,E1 -1916.987,E2 -1916.987} C_VEL
LIN {X 0,Y 580.259,Z 299.2,A -85,B 0,C 180,E1 -1919.774,E2 -1919.774} C_VEL
LIN {X 0,Y 580.275,Z 299.205,A -85,B 0,C 180,E1 -1922.201,E2 -1922.201} C_VEL
LIN {X 0,Y 580.269,Z 299.2,A -85,B 0,C 180,E1 -1924.697,E2 -1924.697} C_VEL
LIN {X 0,Y 580.267,Z 299.2,A -85,B 0,C 180,E1 -1927.27,E2 -1927.27} C_VEL
LIN {X 0,Y 580.278,Z 299.203,A -85,B 0,C 180,E1 -1930.269,E2 -1930.269} C_VEL
LIN {X 0,Y 580.243,Z 299.202,A -85,B 0,C 180,E1 -1932.708,E2 -1932.708} C_VEL
LIN {X 0,Y 580.245,Z 299.202,A -85,B 0,C 180,E1 -1935.611,E2 -1935.611} C_VEL
LIN {X 0,Y 580.245,Z 299.207,A -85,B 0,C 180,E1 -1938.228,E2 -1938.228} C_VEL
LIN {X 0,Y 580.256,Z 299.198,A -85,B 0,C 180,E1 -1940.963,E2 -1940.963} C_VEL
LIN {X 0,Y 580.232,Z 299.201,A -85,B 0,C 180,E1 -1943.594,E2 -1943.594} C_VEL
LIN {X 0,Y 580.27,Z 299.204,A -85,B 0,C 180,E1 -1946.142,E2 -1946.142} C_VEL
LIN {X 0,Y 580.263,Z 299.2,A -85,B 0,C 180,E1 -1948.614,E2 -1948.614} C_VEL
LIN {X 0,Y 580.278,Z 299.196,A -85,B 0,C 180,E1 -1951.023,E2 -1951.023} C_VEL
LIN {X 0,Y 580.244,Z 299.207,A -85,B 0,C 180,E1 -1954.149,E2 -1954.149} C_VEL
LIN {X 0,Y 580.259,Z 299.201,A -85,B 0,C 180,E1 -1956.441,E2 -1956.441} C_VEL
LIN {X 0,Y 580.26,Z 299.201,A -85,B 0,C 180,E1 -1959.437,E2 -1959.437} C_VEL
LIN {X 0,Y 580.241,Z 299.208,A -85,B 0,C 180,E1 -1961.644,E2 -1961.644} C_VEL
LIN {X 0,Y 580.249,Z 299.211,A -85,B 0,C 180,E1 -1963.825,E2 -1963.825} C_VEL
LIN {X 0,Y 580.301,Z 299.199,A -85,B 0,C 180,E1 -1965.982,E2 -1965.982} C_VEL
LIN {X 0,Y 580.296,Z 299.194,A -85,B 0,C 180,E1 -1968.827,E2 -1968.827} C_VEL
LIN {X 0,Y 580.286,Z 299.205,A -85,B 0,C 180,E1 -1971.643,E2 -1971.643} C_VEL
LIN {X 0,Y 580.26,Z 299.208,A -85,B 0,C 180,E1 -1973.742,E2 -1973.742} C_VEL
LIN {X 0,Y 580.246,Z 299.21,A -85,B 0,C 180,E1 -1975.833,E2 -1975.833} C_VEL
LIN {X 0,Y 580.315,Z 299.199,A -85,B 0,C 180,E1 -1977.918,E2 -1977.918} C_VEL
LIN {X 0,Y 580.329,Z 299.194,A -85,B 0,C 180,E1 -1980,E2 -1980} C_VEL
LIN {X 0,Y 580.303,Z 299.194,A -85,B 0,C 180,E1 -1982.777,E2 -1982.777} C_VEL
LIN {X 0,Y 580.302,Z 299.203,A -85,B 0,C 180,E1 -1985.56,E2 -1985.56} C_VEL
LIN {X 0,Y 580.289,Z 299.195,A -85,B 0,C 180,E1 -1988.357,E2 -1988.357} C_VEL
LIN {X 0,Y 580.292,Z 299.199,A -85,B 0,C 180,E1 -1991.191,E2 -1991.191} C_VEL
LIN {X 0,Y 580.285,Z 299.198,A -85,B 0,C 180,E1 -1994.018,E2 -1994.018} C_VEL
LIN {X 0,Y 580.258,Z 299.2,A -85,B 0,C 180,E1 -1996.899,E2 -1996.899} C_VEL
LIN {X 0,Y 580.265,Z 299.203,A -85,B 0,C 180,E1 -1999.824,E2 -1999.824} C_VEL
LIN {X 0,Y 580.276,Z 299.202,A -85,B 0,C 180,E1 -2001.289,E2 -2001.289} C_VEL
LIN {X 0,Y 579.561,Z 299.297,A -85,B 0,C 180,E1 -2001.868,E2 -2001.868} C_VEL
LIN {X 0,Y 576.674,Z 299.657,A -85,B 0,C 180,E1 -2002.808,E2 -2002.808} C_VEL
LIN {X 0,Y 574.273,Z 299.956,A -85,B 0,C 180,E1 -2003.564,E2 -2003.564} C_VEL
LIN {X 0,Y 573.261,Z 300.073,A -85,B 0,C 180,E1 -2004.148,E2 -2004.148} C_VEL
LIN {X 0,Y 573.188,Z 300.081,A -85,B 0,C 180,E1 -2004.345,E2 -2004.345} C_VEL
LIN {X 0,Y 573.184,Z 300.082,A -85,B 0,C 180,E1 -2006.979,E2 -2006.979} C_VEL
LIN {X 0,Y 573.212,Z 300.081,A -85,B 0,C 180,E1 -2009.484,E2 -2009.484} C_VEL
LIN {X 0,Y 573.228,Z 300.075,A -85,B 0,C 180,E1 -2012.226,E2 -2012.226} C_VEL
LIN {X 0,Y 573.213,Z 300.078,A -85,B 0,C 180,E1 -2014.77,E2 -2014.77} C_VEL
LIN {X 0,Y 573.215,Z 300.078,A -85,B 0,C 180,E1 -2017.809,E2 -2017.809} C_VEL
LIN {X 0,Y 573.223,Z 300.074,A -85,B 0,C 180,E1 -2020.527,E2 -2020.527} C_VEL
LIN {X 0,Y 573.203,Z 300.084,A -85,B 0,C 180,E1 -2023.666,E2 -2023.666} C_VEL
LIN {X 0,Y 573.195,Z 300.077,A -85,B 0,C 180,E1 -2026.638,E2 -2026.638} C_VEL
LIN {X 0,Y 573.242,Z 300.083,A -85,B 0,C 180,E1 -2029.476,E2 -2029.476} C_VEL
LIN {X 0,Y 573.211,Z 300.076,A -85,B 0,C 180,E1 -2032.191,E2 -2032.191} C_VEL
LIN {X 0,Y 573.222,Z 300.084,A -85,B 0,C 180,E1 -2035.231,E2 -2035.231} C_VEL
LIN {X 0,Y 573.221,Z 300.076,A -85,B 0,C 180,E1 -2038.184,E2 -2038.184} C_VEL
LIN {X 0,Y 573.229,Z 300.076,A -85,B 0,C 180,E1 -2040.633,E2 -2040.633} C_VEL
LIN {X 0,Y 573.193,Z 300.086,A -85,B 0,C 180,E1 -2043.517,E2 -2043.517} C_VEL
LIN {X 0,Y 573.191,Z 300.081,A -85,B 0,C 180,E1 -2046.133,E2 -2046.133} C_VEL
LIN {X 0,Y 573.245,Z 300.081,A -85,B 0,C 180,E1 -2049.174,E2 -2049.174} C_VEL
LIN {X 0,Y 573.208,Z 300.07,A -85,B 0,C 180,E1 -2052.151,E2 -2052.151} C_VEL
LIN {X 0,Y 573.214,Z 300.087,A -85,B 0,C 180,E1 -2055.08,E2 -2055.08} C_VEL
LIN {X 0,Y 573.276,Z 300.289,A -85,B 0,C 180,E1 -2056.463,E2 -2056.463} C_VEL
LIN {X 0,Y 573.577,Z 301.546,A -85,B 0,C 180,E1 -2056.576,E2 -2056.576} C_VEL
LIN {X 0,Y 574.03,Z 303.572,A -85,B 0,C 180,E1 -2056.616,E2 -2056.616} C_VEL
LIN {X 0,Y 573.911,Z 380.955,A -85,B 0,C 180,E1 -2057.603,E2 -2057.603} C_VEL
LIN {X 0,Y 573.815,Z 394.225,A -85,B 0,C 180,E1 -2057.915,E2 -2057.915} C_VEL
LIN {X 0,Y 573.717,Z 406.383,A -85,B 0,C 180,E1 -2058.339,E2 -2058.339} C_VEL
LIN {X 0,Y 573.611,Z 417.863,A -85,B 0,C 180,E1 -2058.877,E2 -2058.877} C_VEL
LIN {X 0,Y 573.448,Z 429.551,A -85,B 0,C 180,E1 -2059.586,E2 -2059.586} C_VEL
LIN {X 0,Y 573.333,Z 440.07,A -85,B 0,C 180,E1 -2060.386,E2 -2060.386} C_VEL
LIN {X 0,Y 573.241,Z 448.667,A -85,B 0,C 180,E1 -2061.185,E2 -2061.185} C_VEL
LIN {X 0,Y 573.161,Z 456.588,A -85,B 0,C 180,E1 -2062.071,E2 -2062.071} C_VEL
LIN {X 0,Y 573.093,Z 464.524,A -85,B 0,C 180,E1 -2063.163,E2 -2063.163} C_VEL
LIN {X 0,Y 573.071,Z 471.45,A -85,B 0,C 180,E1 -2064.37,E2 -2064.37} C_VEL
LIN {X 0,Y 573.029,Z 476.192,A -85,B 0,C 180,E1 -2065.428,E2 -2065.428} C_VEL
LIN {X 0,Y 573.022,Z 479.825,A -85,B 0,C 180,E1 -2066.484,E2 -2066.484} C_VEL
LIN {X 0,Y 572.959,Z 481.702,A -85,B 0,C 180,E1 -2067.188,E2 -2067.188} C_VEL
LIN {X 0,Y 572.939,Z 483.127,A -85,B 0,C 180,E1 -2067.891,E2 -2067.891} C_VEL
LIN {X 0,Y 572.941,Z 484.756,A -85,B 0,C 180,E1 -2069.297,E2 -2069.297} C_VEL
LIN {X 0,Y 572.939,Z 484.996,A -85,B 0,C 180,E1 -2070,E2 -2070} C_VEL
LIN {X 0,Y 572.94,Z 484.815,A -85,B 0,C 180,E1 -2070.703,E2 -2070.703} C_VEL
LIN {X 0,Y 572.94,Z 483.271,A -85,B 0,C 180,E1 -2072.109,E2 -2072.109} C_VEL
LIN {X 0,Y 572.96,Z 481.91,A -85,B 0,C 180,E1 -2072.812,E2 -2072.812} C_VEL
LIN {X 0,Y 573.015,Z 479.031,A -85,B 0,C 180,E1 -2073.868,E2 -2073.868} C_VEL
LIN {X 0,Y 572.963,Z 475.132,A -85,B 0,C 180,E1 -2074.926,E2 -2074.926} C_VEL
LIN {X 0,Y 573.075,Z 470.1,A -85,B 0,C 180,E1 -2075.983,E2 -2075.983} C_VEL
LIN {X 0,Y 573.083,Z 463.777,A -85,B 0,C 180,E1 -2077.044,E2 -2077.044} C_VEL
LIN {X 0,Y 573.175,Z 455.855,A -85,B 0,C 180,E1 -2078.106,E2 -2078.106} C_VEL
LIN {X 0,Y 573.287,Z 446.004,A -85,B 0,C 180,E1 -2079.17,E2 -2079.17} C_VEL
LIN {X 0,Y 573.426,Z 435.691,A -85,B 0,C 180,E1 -2080.058,E2 -2080.058} C_VEL
LIN {X 0,Y 573.563,Z 424.106,A -85,B 0,C 180,E1 -2080.855,E2 -2080.855} C_VEL
LIN {X 0,Y 573.643,Z 412.496,A -85,B 0,C 180,E1 -2081.483,E2 -2081.483} C_VEL
LIN {X 0,Y 573.758,Z 400.492,A -85,B 0,C 180,E1 -2081.974,E2 -2081.974} C_VEL
LIN {X 0,Y 573.867,Z 387.454,A -85,B 0,C 180,E1 -2082.353,E2 -2082.353} C_VEL
LIN {X 0,Y 573.943,Z 375.107,A -85,B 0,C 180,E1 -2082.576,E2 -2082.576} C_VEL
LIN {X 0,Y 573.98,Z 302.953,A -85,B 0,C 180,E1 -2083.483,E2 -2083.483} C_VEL
LIN {X 0,Y 573.37,Z 300.797,A -85,B 0,C 180,E1 -2083.557,E2 -2083.557} C_VEL
LIN {X 0,Y 573.25,Z 300.113,A -85,B 0,C 180,E1 -2083.696,E2 -2083.696} C_VEL
LIN {X 0,Y 573.213,Z 300.077,A -85,B 0,C 180,E1 -2086.379,E2 -2086.379} C_VEL
LIN {X 0,Y 573.225,Z 300.079,A -85,B 0,C 180,E1 -2089.331,E2 -2089.331} C_VEL
LIN {X 0,Y 573.218,Z 300.076,A -85,B 0,C 180,E1 -2091.581,E2 -2091.581} C_VEL
LIN {X 0,Y 573.188,Z 300.08,A -85,B 0,C 180,E1 -2093.867,E2 -2093.867} C_VEL
LIN {X 0,Y 573.191,Z 300.085,A -85,B 0,C 180,E1 -2096.483,E2 -2096.483} C_VEL
LIN {X 0,Y 573.224,Z 300.077,A -85,B 0,C 180,E1 -2099.368,E2 -2099.368} C_VEL
LIN {X 0,Y 573.228,Z 300.078,A -85,B 0,C 180,E1 -2102.224,E2 -2102.224} C_VEL
LIN {X 0,Y 573.221,Z 300.086,A -85,B 0,C 180,E1 -2104.769,E2 -2104.769} C_VEL
LIN {X 0,Y 573.21,Z 300.076,A -85,B 0,C 180,E1 -2107.809,E2 -2107.809} C_VEL
LIN {X 0,Y 573.242,Z 300.081,A -85,B 0,C 180,E1 -2110.524,E2 -2110.524} C_VEL
LIN {X 0,Y 573.198,Z 300.076,A -85,B 0,C 180,E1 -2113.664,E2 -2113.664} C_VEL
LIN {X 0,Y 573.188,Z 300.091,A -85,B 0,C 180,E1 -2116.636,E2 -2116.636} C_VEL
LIN {X 0,Y 573.223,Z 300.074,A -85,B 0,C 180,E1 -2119.476,E2 -2119.476} C_VEL
LIN {X 0,Y 573.213,Z 300.077,A -85,B 0,C 180,E1 -2122.19,E2 -2122.19} C_VEL
LIN {X 0,Y 573.211,Z 300.079,A -85,B 0,C 180,E1 -2125.231,E2 -2125.231} C_VEL
LIN {X 0,Y 573.228,Z 300.074,A -85,B 0,C 180,E1 -2127.774,E2 -2127.774} C_VEL
LIN {X 0,Y 573.224,Z 300.079,A -85,B 0,C 180,E1 -2130.632,E2 -2130.632} C_VEL
LIN {X 0,Y 573.204,Z 300.077,A -85,B 0,C 180,E1 -2133.512,E2 -2133.512} C_VEL
LIN {X 0,Y 573.184,Z 300.085,A -85,B 0,C 180,E1 -2136.132,E2 -2136.132} C_VEL
LIN {X 0,Y 573.218,Z 300.076,A -85,B 0,C 180,E1 -2139.172,E2 -2139.172} C_VEL
LIN {X 0,Y 573.186,Z 300.081,A -85,B 0,C 180,E1 -2141.41,E2 -2141.41} C_VEL
LIN {X 0,Y 573.202,Z 300.078,A -85,B 0,C 180,E1 -2143.62,E2 -2143.62} C_VEL
LIN {X 0,Y 573.184,Z 300.089,A -85,B 0,C 180,E1 -2146.528,E2 -2146.528} C_VEL
LIN {X 0,Y 573.227,Z 300.075,A -85,B 0,C 180,E1 -2149.403,E2 -2149.403} C_VEL
LIN {X 0,Y 573.227,Z 300.082,A -85,B 0,C 180,E1 -2152.249,E2 -2152.249} C_VEL
LIN {X 0,Y 573.269,Z 300.071,A -85,B 0,C 180,E1 -2155.077,E2 -2155.077} C_VEL
LIN {X 0,Y 573.281,Z 300.071,A -85,B 0,C 180,E1 -2157.892,E2 -2157.892} C_VEL
LIN {X 0,Y 573.318,Z 300.068,A -85,B 0,C 180,E1 -2160.702,E2 -2160.702} C_VEL
LIN {X 0,Y 573.282,Z 300.071,A -85,B 0,C 180,E1 -2162.811,E2 -2162.811} C_VEL
LIN {X 0,Y 573.253,Z 300.072,A -85,B 0,C 180,E1 -2165.629,E2 -2165.629} C_VEL
LIN {X 0,Y 573.203,Z 300.079,A -85,B 0,C 180,E1 -2167.751,E2 -2167.751} C_VEL
LIN {X 0,Y 573.234,Z 300.079,A -85,B 0,C 180,E1 -2170.597,E2 -2170.597} C_VEL
LIN {X 0,Y 573.203,Z 300.077,A -85,B 0,C 180,E1 -2173.471,E2 -2173.471} C_VEL
LIN {X 0,Y 573.209,Z 300.079,A -85,B 0,C 180,E1 -2175.649,E2 -2175.649} C_VEL
LIN {X 0,Y 573.194,Z 300.082,A -85,B 0,C 180,E1 -2178.59,E2 -2178.59} C_VEL
LIN {X 0,Y 573.243,Z 300.07,A -85,B 0,C 180,E1 -2181.291,E2 -2181.291} C_VEL
LIN {X 0,Y 573.206,Z 300.082,A -85,B 0,C 180,E1 -2183.867,E2 -2183.867} C_VEL
LIN {X 0,Y 573.197,Z 300.083,A -85,B 0,C 180,E1 -2186.486,E2 -2186.486} C_VEL
LIN {X 0,Y 573.235,Z 300.073,A -85,B 0,C 180,E1 -2189.368,E2 -2189.368} C_VEL
LIN {X 0,Y 573.241,Z 300.082,A -85,B 0,C 180,E1 -2192.228,E2 -2192.228} C_VEL
LIN {X 0,Y 573.212,Z 300.077,A -85,B 0,C 180,E1 -2194.769,E2 -2194.769} C_VEL
LIN {X 0,Y 573.213,Z 300.083,A -85,B 0,C 180,E1 -2197.809,E2 -2197.809} C_VEL
LIN {X 0,Y 573.24,Z 300.077,A -85,B 0,C 180,E1 -2200.526,E2 -2200.526} C_VEL
LIN {X 0,Y 573.195,Z 300.08,A -85,B 0,C 180,E1 -2203.363,E2 -2203.363} C_VEL
LIN {X 0,Y 573.199,Z 300.084,A -85,B 0,C 180,E1 -2206.336,E2 -2206.336} C_VEL
LIN {X 0,Y 573.242,Z 300.076,A -85,B 0,C 180,E1 -2209.476,E2 -2209.476} C_VEL
LIN {X 0,Y 573.215,Z 300.085,A -85,B 0,C 180,E1 -2212.192,E2 -2212.192} C_VEL
LIN {X 0,Y 573.215,Z 300.078,A -85,B 0,C 180,E1 -2215.232,E2 -2215.232} C_VEL
LIN {X 0,Y 573.228,Z 300.082,A -85,B 0,C 180,E1 -2217.776,E2 -2217.776} C_VEL
LIN {X 0,Y 573.22,Z 300.074,A -85,B 0,C 180,E1 -2220.632,E2 -2220.632} C_VEL
LIN {X 0,Y 573.256,Z 300.226,A -85,B 0,C 180,E1 -2222.852,E2 -2222.852} C_VEL
LIN {X 0,Y 574.603,Z 306.186,A -85,B 0,C 180,E1 -2223.588,E2 -2223.588} C_VEL
LIN {X 0,Y 574.546,Z 328.24,A -85,B 0,C 180,E1 -2226.001,E2 -2226.001} C_VEL
LIN {X 0,Y 574.308,Z 349.052,A -85,B 0,C 180,E1 -2228.293,E2 -2228.293} C_VEL
LIN {X 0,Y 573.993,Z 374.097,A -85,B 0,C 180,E1 -2231.067,E2 -2231.067} C_VEL
LIN {X 0,Y 573.731,Z 399.312,A -85,B 0,C 180,E1 -2233.819,E2 -2233.819} C_VEL
LIN {X 0,Y 573.519,Z 420.898,A -85,B 0,C 180,E1 -2236.13,E2 -2236.13} C_VEL
LIN {X 0,Y 574.078,Z 426.739,A -85,B 0,C 180,E1 -2236.234,E2 -2236.234} C_VEL
LIN {X 0,Y 573.886,Z 530.957,A -85,B 0,C 180,E1 -2237.558,E2 -2237.558} C_VEL
LIN {X 0,Y 573.838,Z 543.464,A -85,B 0,C 180,E1 -2237.848,E2 -2237.848} C_VEL
LIN {X 0,Y 573.7,Z 555.923,A -85,B 0,C 180,E1 -2238.276,E2 -2238.276} C_VEL
LIN {X 0,Y 573.595,Z 567.444,A -85,B 0,C 180,E1 -2238.81,E2 -2238.81} C_VEL
LIN {X 0,Y 573.469,Z 578.913,A -85,B 0,C 180,E1 -2239.497,E2 -2239.497} C_VEL
LIN {X 0,Y 573.345,Z 589.543,A -85,B 0,C 180,E1 -2240.297,E2 -2240.297} C_VEL
